LIN {X 0,Y 470.964,Z 381.158,A -85,B 0,C 180,E1 -7452.523,E2 -7452.523} C_VEL
LIN {X 0,Y 470.095,Z 393.376,A -85,B 0,C 180,E1 -7453.721,E2 -7453.721} C_VEL
LIN {X 0,Y 469.333,Z 404.5,A -85,B 0,C 180,E1 -7455.03,E2 -7455.03} C_VEL
LIN {X 0,Y 468.532,Z 415.308,A -85,B 0,C 180,E1 -7456.556,E2 -7456.556} C_VEL
LIN {X 0,Y 467.988,Z 424.27,A -85,B 0,C 180,E1 -7458.083,E2 -7458.083} C_VEL
LIN {X 0,Y 467.475,Z 431.699,A -85,B 0,C 180,E1 -7459.606,E2 -7459.606} C_VEL
LIN {X 0,Y 467.146,Z 438.641,A -85,B 0,C 180,E1 -7461.347,E2 -7461.347} C_VEL
LIN {X 0,Y 466.909,Z 444.098,A -85,B 0,C 180,E1 -7463.084,E2 -7463.084} C_VEL
LIN {X 0,Y 466.76,Z 448.219,A -85,B 0,C 180,E1 -7464.817,E2 -7464.817} C_VEL
LIN {X 0,Y 466.725,Z 451.115,A -85,B 0,C 180,E1 -7466.547,E2 -7466.547} C_VEL
LIN {X 0,Y 466.632,Z 452.862,A -85,B 0,C 180,E1 -7468.274,E2 -7468.274} C_VEL
LIN {X 0,Y 466.598,Z 453.473,A -85,B 0,C 180,E1 -7470,E2 -7470} C_VEL
LIN {X 0,Y 466.633,Z 452.914,A -85,B 0,C 180,E1 -7471.726,E2 -7471.726} C_VEL
LIN {X 0,Y 466.726,Z 451.237,A -85,B 0,C 180,E1 -7473.453,E2 -7473.453} C_VEL
LIN {X 0,Y 466.754,Z 448.408,A -85,B 0,C 180,E1 -7475.183,E2 -7475.183} C_VEL
LIN {X 0,Y 466.905,Z 444.353,A -85,B 0,C 180,E1 -7476.916,E2 -7476.916} C_VEL
LIN {X 0,Y 467.137,Z 438.975,A -85,B 0,C 180,E1 -7478.653,E2 -7478.653} C_VEL
LIN {X 0,Y 467.457,Z 432.123,A -85,B 0,C 180,E1 -7480.394,E2 -7480.394} C_VEL
LIN {X 0,Y 467.967,Z 424.747,A -85,B 0,C 180,E1 -7481.917,E2 -7481.917} C_VEL
LIN {X 0,Y 468.503,Z 415.866,A -85,B 0,C 180,E1 -7483.445,E2 -7483.445} C_VEL
LIN {X 0,Y 469.115,Z 406.807,A -85,B 0,C 180,E1 -7484.755,E2 -7484.755} C_VEL
LIN {X 0,Y 469.864,Z 396.119,A -85,B 0,C 180,E1 -7486.064,E2 -7486.064} C_VEL
LIN {X 0,Y 470.706,Z 384.762,A -85,B 0,C 180,E1 -7487.232,E2 -7487.232} C_VEL
LIN {X 0,Y 471.57,Z 371.7,A -85,B 0,C 180,E1 -7488.351,E2 -7488.351} C_VEL
LIN {X 0,Y 472.418,Z 357.63,A -85,B 0,C 180,E1 -7489.33,E2 -7489.33} C_VEL
LIN {X 0,Y 473.155,Z 344.313,A -85,B 0,C 180,E1 -7490.07,E2 -7490.07} C_VEL
LIN {X 0,Y 473.771,Z 329.352,A -85,B 0,C 180,E1 -7490.715,E2 -7490.715} C_VEL
LIN {X 0,Y 474.241,Z 315.159,A -85,B 0,C 180,E1 -7491.159,E2 -7491.159} C_VEL
LIN {X 0,Y 474.531,Z 299.207,A -85,B 0,C 180,E1 -7491.481,E2 -7491.481} C_VEL
LIN {X 0,Y 476.095,Z 164.579,A -85,B 0,C 180,E1 -7493.562,E2 -7493.562} C_VEL
LIN {X 0,Y 472.151,Z 147.036,A -85,B 0,C 180,E1 -7494.059,E2 -7494.059} C_VEL
LIN {X 0,Y 471.11,Z 143.654,A -85,B 0,C 180,E1 -7494.183,E2 -7494.183} C_VEL
LIN {X 0,Y 467.58,Z 127.87,A -85,B 0,C 180,E1 -7497.183,E2 -7497.183} C_VEL
LIN {X 0,Y 467.54,Z 127.872,A -85,B 0,C 180,E1 -7500.736,E2 -7500.736} C_VEL
LIN {X 0,Y 467.552,Z 127.869,A -85,B 0,C 180,E1 -7503.791,E2 -7503.791} C_VEL
LIN {X 0,Y 467.499,Z 127.876,A -85,B 0,C 180,E1 -7506.965,E2 -7506.965} C_VEL
LIN {X 0,Y 467.523,Z 127.868,A -85,B 0,C 180,E1 -7509.946,E2 -7509.946} C_VEL
LIN {X 0,Y 467.517,Z 127.874,A -85,B 0,C 180,E1 -7512.568,E2 -7512.568} C_VEL
LIN {X 0,Y 467.563,Z 127.872,A -85,B 0,C 180,E1 -7515.052,E2 -7515.052} C_VEL
LIN {X 0,Y 467.561,Z 127.864,A -85,B 0,C 180,E1 -7518.726,E2 -7518.726} C_VEL
LIN {X 0,Y 467.542,Z 127.863,A -85,B 0,C 180,E1 -7521.953,E2 -7521.953} C_VEL
LIN {X 0,Y 467.552,Z 127.869,A -85,B 0,C 180,E1 -7525.166,E2 -7525.166} C_VEL
LIN {X 0,Y 467.551,Z 127.861,A -85,B 0,C 180,E1 -7528.257,E2 -7528.257} C_VEL
LIN {X 0,Y 467.526,Z 127.869,A -85,B 0,C 180,E1 -7531.247,E2 -7531.247} C_VEL
LIN {X 0,Y 467.58,Z 127.866,A -85,B 0,C 180,E1 -7534.401,E2 -7534.401} C_VEL
LIN {X 0,Y 467.57,Z 127.862,A -85,B 0,C 180,E1 -7536.995,E2 -7536.995} C_VEL
LIN {X 0,Y 467.613,Z 127.861,A -85,B 0,C 180,E1 -7539.777,E2 -7539.777} C_VEL
LIN {X 0,Y 467.568,Z 127.867,A -85,B 0,C 180,E1 -7542.505,E2 -7542.505} C_VEL
LIN {X 0,Y 467.597,Z 127.86,A -85,B 0,C 180,E1 -7545.196,E2 -7545.196} C_VEL
LIN {X 0,Y 467.66,Z 127.857,A -85,B 0,C 180,E1 -7547.855,E2 -7547.855} C_VEL
LIN {X 0,Y 467.66,Z 127.849,A -85,B 0,C 180,E1 -7551.357,E2 -7551.357} C_VEL
LIN {X 0,Y 467.706,Z 127.85,A -85,B 0,C 180,E1 -7553.962,E2 -7553.962} C_VEL
LIN {X 0,Y 467.816,Z 127.836,A -85,B 0,C 180,E1 -7557.417,E2 -7557.417} C_VEL
LIN {X 0,Y 467.855,Z 127.828,A -85,B 0,C 180,E1 -7560,E2 -7560} C_VEL
LIN {X 0,Y 467.852,Z 127.829,A -85,B 0,C 180,E1 -7562.583,E2 -7562.583} C_VEL
LIN {X 0,Y 467.715,Z 127.847,A -85,B 0,C 180,E1 -7566.038,E2 -7566.038} C_VEL
LIN {X 0,Y 467.67,Z 127.85,A -85,B 0,C 180,E1 -7568.643,E2 -7568.643} C_VEL
LIN {X 0,Y 467.659,Z 127.853,A -85,B 0,C 180,E1 -7572.145,E2 -7572.145} C_VEL
LIN {X 0,Y 467.651,Z 127.856,A -85,B 0,C 180,E1 -7575.884,E2 -7575.884} C_VEL
LIN {X 0,Y 467.624,Z 127.864,A -85,B 0,C 180,E1 -7579.308,E2 -7579.308} C_VEL
LIN {X 0,Y 467.536,Z 127.866,A -85,B 0,C 180,E1 -7582.074,E2 -7582.074} C_VEL
LIN {X 0,Y 467.57,Z 127.871,A -85,B 0,C 180,E1 -7584.889,E2 -7584.889} C_VEL
LIN {X 0,Y 467.582,Z 127.863,A -85,B 0,C 180,E1 -7587.771,E2 -7587.771} C_VEL
LIN {X 0,Y 467.569,Z 127.868,A -85,B 0,C 180,E1 -7591.044,E2 -7591.044} C_VEL
LIN {X 0,Y 467.579,Z 127.862,A -85,B 0,C 180,E1 -7594.24,E2 -7594.24} C_VEL
LIN {X 0,Y 467.549,Z 127.867,A -85,B 0,C 180,E1 -7597.186,E2 -7597.186} C_VEL
LIN {X 0,Y 467.576,Z 127.866,A -85,B 0,C 180,E1 -7600.265,E2 -7600.265} C_VEL
LIN {X 0,Y 467.588,Z 127.866,A -85,B 0,C 180,E1 -7602.567,E2 -7602.567} C_VEL
LIN {X 0,Y 467.567,Z 127.865,A -85,B 0,C 180,E1 -7605.052,E2 -7605.052} C_VEL
LIN {X 0,Y 467.59,Z 127.861,A -85,B 0,C 180,E1 -7607.44,E2 -7607.44} C_VEL
LIN {X 0,Y 467.583,Z 127.863,A -85,B 0,C 180,E1 -7610.855,E2 -7610.855} C_VEL
LIN {X 0,Y 467.561,Z 127.871,A -85,B 0,C 180,E1 -7614.261,E2 -7614.261} C_VEL
LIN {X 0,Y 467.583,Z 127.866,A -85,B 0,C 180,E1 -7617.321,E2 -7617.321} C_VEL
LIN {X 0,Y 467.577,Z 127.992,A -85,B 0,C 180,E1 -7619.641,E2 -7619.641} C_VEL
LIN {X 0,Y 471.398,Z 143.466,A -85,B 0,C 180,E1 -7622.297,E2 -7622.297} C_VEL
LIN {X 0,Y 472.18,Z 147.627,A -85,B 0,C 180,E1 -7622.979,E2 -7622.979} C_VEL
LIN {X 0,Y 471.23,Z 165.357,A -85,B 0,C 180,E1 -7625.608,E2 -7625.608} C_VEL
LIN {X 0,Y 471.125,Z 167.06,A -85,B 0,C 180,E1 -7625.858,E2 -7625.858} C_VEL
LIN {X 0,Y 475.883,Z 191.887,A -85,B 0,C 180,E1 -7626.518,E2 -7626.518} C_VEL
LIN {X 0,Y 474.175,Z 334.044,A -85,B 0,C 180,E1 -7628.736,E2 -7628.736} C_VEL
LIN {X 0,Y 473.612,Z 349.775,A -85,B 0,C 180,E1 -7629.159,E2 -7629.159} C_VEL
LIN {X 0,Y 473.059,Z 363.831,A -85,B 0,C 180,E1 -7629.704,E2 -7629.704} C_VEL
LIN {X 0,Y 472.272,Z 378.294,A -85,B 0,C 180,E1 -7630.438,E2 -7630.438} C_VEL
LIN {X 0,Y 471.417,Z 391.803,A -85,B 0,C 180,E1 -7631.305,E2 -7631.305} C_VEL
LIN {X 0,Y 470.502,Z 405.559,A -85,B 0,C 180,E1 -7632.393,E2 -7632.393} C_VEL
LIN {X 0,Y 469.702,Z 418.015,A -85,B 0,C 180,E1 -7633.595,E2 -7633.595} C_VEL
LIN {X 0,Y 468.789,Z 430.23,A -85,B 0,C 180,E1 -7635.012,E2 -7635.012} C_VEL
LIN {X 0,Y 468.08,Z 441.095,A -85,B 0,C 180,E1 -7636.542,E2 -7636.542} C_VEL
LIN {X 0,Y 467.611,Z 450.148,A -85,B 0,C 180,E1 -7638.073,E2 -7638.073} C_VEL
LIN {X 0,Y 467.228,Z 457.657,A -85,B 0,C 180,E1 -7639.601,E2 -7639.601} C_VEL
LIN {X 0,Y 466.908,Z 464.664,A -85,B 0,C 180,E1 -7641.343,E2 -7641.343} C_VEL
LIN {X 0,Y 466.818,Z 470.178,A -85,B 0,C 180,E1 -7643.082,E2 -7643.082} C_VEL
LIN {X 0,Y 466.685,Z 474.344,A -85,B 0,C 180,E1 -7644.816,E2 -7644.816} C_VEL
LIN {X 0,Y 466.634,Z 477.265,A -85,B 0,C 180,E1 -7646.546,E2 -7646.546} C_VEL
LIN {X 0,Y 466.604,Z 479.007,A -85,B 0,C 180,E1 -7648.274,E2 -7648.274} C_VEL
LIN {X 0,Y 466.596,Z 479.605,A -85,B 0,C 180,E1 -7650,E2 -7650} C_VEL
LIN {X 0,Y 466.604,Z 479.005,A -85,B 0,C 180,E1 -7651.726,E2 -7651.726} C_VEL
LIN {X 0,Y 466.634,Z 477.259,A -85,B 0,C 180,E1 -7653.454,E2 -7653.454} C_VEL
LIN {X 0,Y 466.686,Z 474.34,A -85,B 0,C 180,E1 -7655.184,E2 -7655.184} C_VEL
LIN {X 0,Y 466.818,Z 470.179,A -85,B 0,C 180,E1 -7656.918,E2 -7656.918} C_VEL
LIN {X 0,Y 466.908,Z 464.662,A -85,B 0,C 180,E1 -7658.657,E2 -7658.657} C_VEL
LIN {X 0,Y 467.227,Z 457.646,A -85,B 0,C 180,E1 -7660.399,E2 -7660.399} C_VEL
LIN {X 0,Y 467.608,Z 450.138,A -85,B 0,C 180,E1 -7661.927,E2 -7661.927} C_VEL
LIN {X 0,Y 468.08,Z 441.088,A -85,B 0,C 180,E1 -7663.458,E2 -7663.458} C_VEL
LIN {X 0,Y 468.789,Z 430.218,A -85,B 0,C 180,E1 -7664.988,E2 -7664.988} C_VEL
LIN {X 0,Y 469.675,Z 418.004,A -85,B 0,C 180,E1 -7666.406,E2 -7666.406} C_VEL
LIN {X 0,Y 470.499,Z 405.548,A -85,B 0,C 180,E1 -7667.607,E2 -7667.607} C_VEL
LIN {X 0,Y 471.406,Z 391.772,A -85,B 0,C 180,E1 -7668.695,E2 -7668.695} C_VEL
LIN {X 0,Y 472.268,Z 378.248,A -85,B 0,C 180,E1 -7669.562,E2 -7669.562} C_VEL
LIN {X 0,Y 473.057,Z 363.696,A -85,B 0,C 180,E1 -7670.301,E2 -7670.301} C_VEL
LIN {X 0,Y 473.673,Z 349.107,A -85,B 0,C 180,E1 -7670.861,E2 -7670.861} C_VEL
LIN {X 0,Y 474.164,Z 333.95,A -85,B 0,C 180,E1 -7671.264,E2 -7671.264} C_VEL
LIN {X 0,Y 475.8,Z 200.78,A -85,B 0,C 180,E1 -7673.34,E2 -7673.34} C_VEL
LIN {X 0,Y 475.737,Z 190.572,A -85,B 0,C 180,E1 -7673.507,E2 -7673.507} C_VEL
LIN {X 0,Y 471.132,Z 167.042,A -85,B 0,C 180,E1 -7674.14,E2 -7674.14} C_VEL
LIN {X 0,Y 472.175,Z 147.582,A -85,B 0,C 180,E1 -7677.024,E2 -7677.024} C_VEL
LIN {X 0,Y 469.786,Z 136.715,A -85,B 0,C 180,E1 -7678.839,E2 -7678.839} C_VEL
LIN {X 0,Y 467.58,Z 127.866,A -85,B 0,C 180,E1 -7680.389,E2 -7680.389} C_VEL
LIN {X 0,Y 467.587,Z 127.862,A -85,B 0,C 180,E1 -7683.788,E2 -7683.788} C_VEL
LIN {X 0,Y 467.549,Z 127.868,A -85,B 0,C 180,E1 -7687.186,E2 -7687.186} C_VEL
LIN {X 0,Y 467.578,Z 127.865,A -85,B 0,C 180,E1 -7690.265,E2 -7690.265} C_VEL
LIN {X 0,Y 467.587,Z 127.861,A -85,B 0,C 180,E1 -7692.567,E2 -7692.567} C_VEL
LIN {X 0,Y 467.567,Z 127.864,A -85,B 0,C 180,E1 -7695.053,E2 -7695.053} C_VEL
LIN {X 0,Y 467.59,Z 127.865,A -85,B 0,C 180,E1 -7697.44,E2 -7697.44} C_VEL
LIN {X 0,Y 467.561,Z 127.866,A -85,B 0,C 180,E1 -7700.853,E2 -7700.853} C_VEL
LIN {X 0,Y 467.56,Z 127.862,A -85,B 0,C 180,E1 -7704.261,E2 -7704.261} C_VEL
LIN {X 0,Y 467.581,Z 127.865,A -85,B 0,C 180,E1 -7707.322,E2 -7707.322} C_VEL
LIN {X 0,Y 467.57,Z 127.863,A -85,B 0,C 180,E1 -7710.668,E2 -7710.668} C_VEL
LIN {X 0,Y 467.588,Z 127.865,A -85,B 0,C 180,E1 -7713.198,E2 -7713.198} C_VEL
LIN {X 0,Y 467.591,Z 127.861,A -85,B 0,C 180,E1 -7716.47,E2 -7716.47} C_VEL
LIN {X 0,Y 467.623,Z 127.854,A -85,B 0,C 180,E1 -7719.777,E2 -7719.777} C_VEL
LIN {X 0,Y 467.597,Z 127.864,A -85,B 0,C 180,E1 -7722.506,E2 -7722.506} C_VEL
LIN {X 0,Y 467.605,Z 127.863,A -85,B 0,C 180,E1 -7725.197,E2 -7725.197} C_VEL
LIN {X 0,Y 467.659,Z 127.849,A -85,B 0,C 180,E1 -7727.855,E2 -7727.855} C_VEL
LIN {X 0,Y 467.67,Z 127.848,A -85,B 0,C 180,E1 -7731.357,E2 -7731.357} C_VEL
LIN {X 0,Y 467.715,Z 127.847,A -85,B 0,C 180,E1 -7733.962,E2 -7733.962} C_VEL
LIN {X 0,Y 467.852,Z 127.828,A -85,B 0,C 180,E1 -7737.417,E2 -7737.417} C_VEL
LIN {X 0,Y 467.855,Z 127.83,A -85,B 0,C 180,E1 -7740,E2 -7740} C_VEL
LIN {X 0,Y 467.817,Z 127.837,A -85,B 0,C 180,E1 -7742.583,E2 -7742.583} C_VEL
LIN {X 0,Y 467.712,Z 127.849,A -85,B 0,C 180,E1 -7746.038,E2 -7746.038} C_VEL
LIN {X 0,Y 467.66,Z 127.851,A -85,B 0,C 180,E1 -7748.643,E2 -7748.643} C_VEL
LIN {X 0,Y 467.659,Z 127.856,A -85,B 0,C 180,E1 -7752.145,E2 -7752.145} C_VEL
LIN {X 0,Y 467.615,Z 127.863,A -85,B 0,C 180,E1 -7755.696,E2 -7755.696} C_VEL
LIN {X 0,Y 467.62,Z 127.859,A -85,B 0,C 180,E1 -7759.308,E2 -7759.308} C_VEL
LIN {X 0,Y 467.535,Z 127.873,A -85,B 0,C 180,E1 -7762.074,E2 -7762.074} C_VEL
LIN {X 0,Y 467.561,Z 127.862,A -85,B 0,C 180,E1 -7764.89,E2 -7764.89} C_VEL
LIN {X 0,Y 467.547,Z 127.865,A -85,B 0,C 180,E1 -7767.774,E2 -7767.774} C_VEL
LIN {X 0,Y 467.549,Z 127.868,A -85,B 0,C 180,E1 -7771.04,E2 -7771.04} C_VEL
LIN {X 0,Y 467.577,Z 127.86,A -85,B 0,C 180,E1 -7774.24,E2 -7774.24} C_VEL
LIN {X 0,Y 467.539,Z 127.871,A -85,B 0,C 180,E1 -7777.184,E2 -7777.184} C_VEL
LIN {X 0,Y 467.557,Z 127.864,A -85,B 0,C 180,E1 -7780.267,E2 -7780.267} C_VEL
LIN {X 0,Y 467.545,Z 127.867,A -85,B 0,C 180,E1 -7783.746,E2 -7783.746} C_VEL
LIN {X 0,Y 467.545,Z 127.867,A -85,B 0,C 180,E1 -7786.254,E2 -7786.254} C_VEL
LIN {X 0,Y 467.556,Z 127.868,A -85,B 0,C 180,E1 -7789.733,E2 -7789.733} C_VEL
LIN {X 0,Y 467.517,Z 127.877,A -85,B 0,C 180,E1 -7792.819,E2 -7792.819} C_VEL
LIN {X 0,Y 467.565,Z 127.867,A -85,B 0,C 180,E1 -7795.762,E2 -7795.762} C_VEL
LIN {X 0,Y 467.527,Z 127.867,A -85,B 0,C 180,E1 -7798.964,E2 -7798.964} C_VEL
LIN {X 0,Y 467.538,Z 127.873,A -85,B 0,C 180,E1 -7802.226,E2 -7802.226} C_VEL
LIN {X 0,Y 467.586,Z 127.922,A -85,B 0,C 180,E1 -7802.927,E2 -7802.927} C_VEL
LIN {X 0,Y 470.737,Z 142.01,A -85,B 0,C 180,E1 -7805.605,E2 -7805.605} C_VEL
LIN {X 0,Y 471.126,Z 143.896,A -85,B 0,C 180,E1 -7805.927,E2 -7805.927} C_VEL
LIN {X 0,Y 472.934,Z 150.367,A -85,B 0,C 180,E1 -7806.132,E2 -7806.132} C_VEL
LIN {X 0,Y 476.111,Z 164.515,A -85,B 0,C 180,E1 -7806.531,E2 -7806.531} C_VEL
LIN {X 0,Y 475.725,Z 202.904,A -85,B 0,C 180,E1 -7807.129,E2 -7807.129} C_VEL
LIN {X 0,Y 475.079,Z 208.751,A -85,B 0,C 180,E1 -7807.19,E2 -7807.19} C_VEL
LIN {X 0,Y 469.531,Z 227.805,A -85,B 0,C 180,E1 -7807.213,E2 -7807.213} C_VEL
LIN {X 0,Y 468.741,Z 233.659,A -85,B 0,C 180,E1 -7807.267,E2 -7807.267} C_VEL
LIN {X 0,Y 467.779,Z 308.963,A -85,B 0,C 180,E1 -7808.466,E2 -7808.466} C_VEL
LIN {X 0,Y 467.327,Z 324.475,A -85,B 0,C 180,E1 -7808.887,E2 -7808.887} C_VEL
LIN {X 0,Y 466.807,Z 338.824,A -85,B 0,C 180,E1 -7809.451,E2 -7809.451} C_VEL
LIN {X 0,Y 466.013,Z 352.734,A -85,B 0,C 180,E1 -7810.164,E2 -7810.164} C_VEL
LIN {X 0,Y 465.186,Z 366.326,A -85,B 0,C 180,E1 -7811.045,E2 -7811.045} C_VEL
LIN {X 0,Y 464.329,Z 378.821,A -85,B 0,C 180,E1 -7812.038,E2 -7812.038} C_VEL
LIN {X 0,Y 463.397,Z 391.471,A -85,B 0,C 180,E1 -7813.252,E2 -7813.252} C_VEL
LIN {X 0,Y 462.548,Z 402.936,A -85,B 0,C 180,E1 -7814.58,E2 -7814.58} C_VEL
LIN {X 0,Y 461.825,Z 412.582,A -85,B 0,C 180,E1 -7815.908,E2 -7815.908} C_VEL
LIN {X 0,Y 461.063,Z 422.108,A -85,B 0,C 180,E1 -7817.468,E2 -7817.468} C_VEL
LIN {X 0,Y 460.627,Z 429.9,A -85,B 0,C 180,E1 -7819.005,E2 -7819.005} C_VEL
LIN {X 0,Y 460.165,Z 437.243,A -85,B 0,C 180,E1 -7820.772,E2 -7820.772} C_VEL
LIN {X 0,Y 459.9,Z 443.069,A -85,B 0,C 180,E1 -7822.537,E2 -7822.537} C_VEL
LIN {X 0,Y 459.817,Z 446.516,A -85,B 0,C 180,E1 -7823.858,E2 -7823.858} C_VEL
LIN {X 0,Y 459.595,Z 450.016,A -85,B 0,C 180,E1 -7825.615,E2 -7825.615} C_VEL
LIN {X 0,Y 459.6,Z 452.328,A -85,B 0,C 180,E1 -7827.371,E2 -7827.371} C_VEL
LIN {X 0,Y 459.521,Z 453.514,A -85,B 0,C 180,E1 -7829.124,E2 -7829.124} C_VEL
LIN {X 0,Y 459.521,Z 453.531,A -85,B 0,C 180,E1 -7830.876,E2 -7830.876} C_VEL
LIN {X 0,Y 459.601,Z 452.415,A -85,B 0,C 180,E1 -7832.629,E2 -7832.629} C_VEL
LIN {X 0,Y 459.594,Z 450.171,A -85,B 0,C 180,E1 -7834.385,E2 -7834.385} C_VEL
LIN {X 0,Y 459.787,Z 446.735,A -85,B 0,C 180,E1 -7836.142,E2 -7836.142} C_VEL
LIN {X 0,Y 459.965,Z 442.035,A -85,B 0,C 180,E1 -7837.904,E2 -7837.904} C_VEL
LIN {X 0,Y 460.255,Z 435.944,A -85,B 0,C 180,E1 -7839.67,E2 -7839.67} C_VEL
LIN {X 0,Y 460.814,Z 428.268,A -85,B 0,C 180,E1 -7841.436,E2 -7841.436} C_VEL
LIN {X 0,Y 461.285,Z 420.112,A -85,B 0,C 180,E1 -7842.983,E2 -7842.983} C_VEL
LIN {X 0,Y 461.986,Z 410.229,A -85,B 0,C 180,E1 -7844.537,E2 -7844.537} C_VEL
LIN {X 0,Y 462.757,Z 400.117,A -85,B 0,C 180,E1 -7845.865,E2 -7845.865} C_VEL
LIN {X 0,Y 463.621,Z 389.042,A -85,B 0,C 180,E1 -7847.09,E2 -7847.09} C_VEL
LIN {X 0,Y 464.406,Z 377.289,A -85,B 0,C 180,E1 -7848.187,E2 -7848.187} C_VEL
LIN {X 0,Y 465.322,Z 364.457,A -85,B 0,C 180,E1 -7849.178,E2 -7849.178} C_VEL
LIN {X 0,Y 466.18,Z 350.381,A -85,B 0,C 180,E1 -7850.058,E2 -7850.058} C_VEL
LIN {X 0,Y 466.925,Z 335.079,A -85,B 0,C 180,E1 -7850.802,E2 -7850.802} C_VEL
LIN {X 0,Y 467.481,Z 319.758,A -85,B 0,C 180,E1 -7851.349,E2 -7851.349} C_VEL
LIN {X 0,Y 467.889,Z 304.527,A -85,B 0,C 180,E1 -7851.708,E2 -7851.708} C_VEL
LIN {X 0,Y 469.572,Z 164.991,A -85,B 0,C 180,E1 -7853.906,E2 -7853.906} C_VEL
LIN {X 0,Y 465.333,Z 147.428,A -85,B 0,C 180,E1 -7854.431,E2 -7854.431} C_VEL
LIN {X 0,Y 463.967,Z 143.875,A -85,B 0,C 180,E1 -7854.577,E2 -7854.577} C_VEL
LIN {X 0,Y 460.858,Z 130.147,A -85,B 0,C 180,E1 -7857.226,E2 -7857.226} C_VEL
LIN {X 0,Y 460.511,Z 128.75,A -85,B 0,C 180,E1 -7857.527,E2 -7857.527} C_VEL
LIN {X 0,Y 460.479,Z 128.751,A -85,B 0,C 180,E1 -7860.243,E2 -7860.243} C_VEL
LIN {X 0,Y 460.501,Z 128.751,A -85,B 0,C 180,E1 -7863.327,E2 -7863.327} C_VEL
LIN {X 0,Y 460.455,Z 128.752,A -85,B 0,C 180,E1 -7866.532,E2 -7866.532} C_VEL
LIN {X 0,Y 460.475,Z 128.746,A -85,B 0,C 180,E1 -7869.869,E2 -7869.869} C_VEL
LIN {X 0,Y 460.457,Z 128.756,A -85,B 0,C 180,E1 -7872.893,E2 -7872.893} C_VEL
LIN {X 0,Y 460.495,Z 128.746,A -85,B 0,C 180,E1 -7875.833,E2 -7875.833} C_VEL
LIN {X 0,Y 460.515,Z 128.746,A -85,B 0,C 180,E1 -7878.987,E2 -7878.987} C_VEL
LIN {X 0,Y 460.484,Z 128.742,A -85,B 0,C 180,E1 -7882.375,E2 -7882.375} C_VEL
LIN {X 0,Y 460.535,Z 128.741,A -85,B 0,C 180,E1 -7885.623,E2 -7885.623} C_VEL
LIN {X 0,Y 460.506,Z 128.735,A -85,B 0,C 180,E1 -7888.742,E2 -7888.742} C_VEL
LIN {X 0,Y 460.498,Z 128.745,A -85,B 0,C 180,E1 -7891.763,E2 -7891.763} C_VEL
LIN {X 0,Y 460.524,Z 128.745,A -85,B 0,C 180,E1 -7894.703,E2 -7894.703} C_VEL
LIN {X 0,Y 460.505,Z 128.742,A -85,B 0,C 180,E1 -7897.571,E2 -7897.571} C_VEL
LIN {X 0,Y 460.564,Z 128.74,A -85,B 0,C 180,E1 -7900.384,E2 -7900.384} C_VEL
LIN {X 0,Y 460.569,Z 128.743,A -85,B 0,C 180,E1 -7904.058,E2 -7904.058} C_VEL
LIN {X 0,Y 460.613,Z 128.732,A -85,B 0,C 180,E1 -7907.666,E2 -7907.666} C_VEL
LIN {X 0,Y 460.612,Z 128.726,A -85,B 0,C 180,E1 -7911.223,E2 -7911.223} C_VEL
LIN {X 0,Y 460.672,Z 128.728,A -85,B 0,C 180,E1 -7913.869,E2 -7913.869} C_VEL
LIN {X 0,Y 460.76,Z 128.715,A -85,B 0,C 180,E1 -7917.377,E2 -7917.377} C_VEL
LIN {X 0,Y 460.825,Z 128.704,A -85,B 0,C 180,E1 -7920,E2 -7920} C_VEL
LIN {X 0,Y 460.792,Z 128.708,A -85,B 0,C 180,E1 -7922.622,E2 -7922.622} C_VEL
LIN {X 0,Y 460.68,Z 128.723,A -85,B 0,C 180,E1 -7926.13,E2 -7926.13} C_VEL
LIN {X 0,Y 460.62,Z 128.729,A -85,B 0,C 180,E1 -7928.776,E2 -7928.776} C_VEL
LIN {X 0,Y 460.612,Z 128.731,A -85,B 0,C 180,E1 -7932.334,E2 -7932.334} C_VEL
LIN {X 0,Y 460.603,Z 128.733,A -85,B 0,C 180,E1 -7935.997,E2 -7935.997} C_VEL
LIN {X 0,Y 460.57,Z 128.739,A -85,B 0,C 180,E1 -7939.615,E2 -7939.615} C_VEL
LIN {X 0,Y 460.512,Z 128.743,A -85,B 0,C 180,E1 -7942.428,E2 -7942.428} C_VEL
LIN {X 0,Y 460.549,Z 128.737,A -85,B 0,C 180,E1 -7945.796,E2 -7945.796} C_VEL
LIN {X 0,Y 460.529,Z 128.743,A -85,B 0,C 180,E1 -7948.234,E2 -7948.234} C_VEL
LIN {X 0,Y 460.522,Z 128.744,A -85,B 0,C 180,E1 -7951.283,E2 -7951.283} C_VEL
LIN {X 0,Y 460.525,Z 128.743,A -85,B 0,C 180,E1 -7954.504,E2 -7954.504} C_VEL
LIN {X 0,Y 460.502,Z 128.743,A -85,B 0,C 180,E1 -7957.623,E2 -7957.623} C_VEL
LIN {X 0,Y 460.54,Z 128.742,A -85,B 0,C 180,E1 -7960.269,E2 -7960.269} C_VEL
LIN {X 0,Y 460.5,Z 128.746,A -85,B 0,C 180,E1 -7963.375,E2 -7963.375} C_VEL
LIN {X 0,Y 460.5,Z 128.747,A -85,B 0,C 180,E1 -7966.624,E2 -7966.624} C_VEL
LIN {X 0,Y 460.543,Z 128.735,A -85,B 0,C 180,E1 -7969.73,E2 -7969.73} C_VEL
LIN {X 0,Y 460.501,Z 128.748,A -85,B 0,C 180,E1 -7972.524,E2 -7972.524} C_VEL
LIN {X 0,Y 460.547,Z 128.744,A -85,B 0,C 180,E1 -7975.624,E2 -7975.624} C_VEL
LIN {X 0,Y 460.538,Z 128.744,A -85,B 0,C 180,E1 -7978.744,E2 -7978.744} C_VEL
LIN {X 0,Y 460.534,Z 128.783,A -85,B 0,C 180,E1 -7979.286,E2 -7979.286} C_VEL
LIN {X 0,Y 464.382,Z 144.41,A -85,B 0,C 180,E1 -7982.02,E2 -7982.02} C_VEL
LIN {X 0,Y 465.346,Z 149.156,A -85,B 0,C 180,E1 -7982.816,E2 -7982.816} C_VEL
LIN {X 0,Y 464.468,Z 165.058,A -85,B 0,C 180,E1 -7985.213,E2 -7985.213} C_VEL
LIN {X 0,Y 464.367,Z 166.838,A -85,B 0,C 180,E1 -7985.481,E2 -7985.481} C_VEL
LIN {X 0,Y 469.365,Z 192.662,A -85,B 0,C 180,E1 -7986.188,E2 -7986.188} C_VEL
LIN {X 0,Y 467.572,Z 333.856,A -85,B 0,C 180,E1 -7988.421,E2 -7988.421} C_VEL
LIN {X 0,Y 466.98,Z 349.574,A -85,B 0,C 180,E1 -7988.849,E2 -7988.849} C_VEL
LIN {X 0,Y 466.363,Z 364.228,A -85,B 0,C 180,E1 -7989.428,E2 -7989.428} C_VEL
LIN {X 0,Y 465.545,Z 378.099,A -85,B 0,C 180,E1 -7990.143,E2 -7990.143} C_VEL
LIN {X 0,Y 464.669,Z 391.607,A -85,B 0,C 180,E1 -7991.023,E2 -7991.023} C_VEL
LIN {X 0,Y 463.678,Z 405.362,A -85,B 0,C 180,E1 -7992.126,E2 -7992.126} C_VEL
LIN {X 0,Y 462.833,Z 417.817,A -85,B 0,C 180,E1 -7993.345,E2 -7993.345} C_VEL
LIN {X 0,Y 461.857,Z 430.031,A -85,B 0,C 180,E1 -7994.782,E2 -7994.782} C_VEL
LIN {X 0,Y 461.119,Z 440.896,A -85,B 0,C 180,E1 -7996.335,E2 -7996.335} C_VEL
LIN {X 0,Y 460.591,Z 449.948,A -85,B 0,C 180,E1 -7997.889,E2 -7997.889} C_VEL
LIN {X 0,Y 460.216,Z 457.458,A -85,B 0,C 180,E1 -7999.441,E2 -7999.441} C_VEL
LIN {X 0,Y 459.851,Z 464.465,A -85,B 0,C 180,E1 -8001.209,E2 -8001.209} C_VEL
LIN {X 0,Y 459.727,Z 469.978,A -85,B 0,C 180,E1 -8002.975,E2 -8002.975} C_VEL
LIN {X 0,Y 459.595,Z 474.145,A -85,B 0,C 180,E1 -8004.736,E2 -8004.736} C_VEL
LIN {X 0,Y 459.53,Z 477.066,A -85,B 0,C 180,E1 -8006.493,E2 -8006.493} C_VEL
LIN {X 0,Y 459.517,Z 478.809,A -85,B 0,C 180,E1 -8008.247,E2 -8008.247} C_VEL
LIN {X 0,Y 459.527,Z 479.407,A -85,B 0,C 180,E1 -8010,E2 -8010} C_VEL
LIN {X 0,Y 459.517,Z 478.806,A -85,B 0,C 180,E1 -8011.753,E2 -8011.753} C_VEL
LIN {X 0,Y 459.53,Z 477.059,A -85,B 0,C 180,E1 -8013.507,E2 -8013.507} C_VEL
LIN {X 0,Y 459.598,Z 474.14,A -85,B 0,C 180,E1 -8015.264,E2 -8015.264} C_VEL
LIN {X 0,Y 459.727,Z 469.979,A -85,B 0,C 180,E1 -8017.025,E2 -8017.025} C_VEL
LIN {X 0,Y 459.851,Z 464.461,A -85,B 0,C 180,E1 -8018.791,E2 -8018.791} C_VEL
LIN {X 0,Y 460.214,Z 457.445,A -85,B 0,C 180,E1 -8020.559,E2 -8020.559} C_VEL
LIN {X 0,Y 460.584,Z 449.936,A -85,B 0,C 180,E1 -8022.111,E2 -8022.111} C_VEL
LIN {X 0,Y 461.119,Z 440.886,A -85,B 0,C 180,E1 -8023.665,E2 -8023.665} C_VEL
LIN {X 0,Y 461.855,Z 430.015,A -85,B 0,C 180,E1 -8025.218,E2 -8025.218} C_VEL
LIN {X 0,Y 462.811,Z 417.801,A -85,B 0,C 180,E1 -8026.656,E2 -8026.656} C_VEL
LIN {X 0,Y 463.679,Z 405.345,A -85,B 0,C 180,E1 -8027.874,E2 -8027.874} C_VEL
LIN {X 0,Y 464.644,Z 391.568,A -85,B 0,C 180,E1 -8028.978,E2 -8028.978} C_VEL
LIN {X 0,Y 465.533,Z 378.043,A -85,B 0,C 180,E1 -8029.857,E2 -8029.857} C_VEL
LIN {X 0,Y 466.352,Z 364.112,A -85,B 0,C 180,E1 -8030.576,E2 -8030.576} C_VEL
LIN {X 0,Y 467.051,Z 348.901,A -85,B 0,C 180,E1 -8031.17,E2 -8031.17} C_VEL
LIN {X 0,Y 467.556,Z 333.74,A -85,B 0,C 180,E1 -8031.58,E2 -8031.58} C_VEL
LIN {X 0,Y 469.117,Z 211.55,A -85,B 0,C 180,E1 -8033.513,E2 -8033.513} C_VEL
LIN {X 0,Y 469.296,Z 191.977,A -85,B 0,C 180,E1 -8033.823,E2 -8033.823} C_VEL
LIN {X 0,Y 464.378,Z 166.694,A -85,B 0,C 180,E1 -8034.535,E2 -8034.535} C_VEL
LIN {X 0,Y 465.34,Z 149.118,A -85,B 0,C 180,E1 -8037.185,E2 -8037.185} C_VEL
LIN {X 0,Y 462.31,Z 135.727,A -85,B 0,C 180,E1 -8039.474,E2 -8039.474} C_VEL
LIN {X 0,Y 460.547,Z 128.742,A -85,B 0,C 180,E1 -8040.745,E2 -8040.745} C_VEL
LIN {X 0,Y 460.53,Z 128.736,A -85,B 0,C 180,E1 -8043.325,E2 -8043.325} C_VEL
LIN {X 0,Y 460.477,Z 128.75,A -85,B 0,C 180,E1 -8046.53,E2 -8046.53} C_VEL
LIN {X 0,Y 460.559,Z 128.744,A -85,B 0,C 180,E1 -8049.86,E2 -8049.86} C_VEL
LIN {X 0,Y 460.513,Z 128.743,A -85,B 0,C 180,E1 -8052.9,E2 -8052.9} C_VEL
LIN {X 0,Y 460.51,Z 128.748,A -85,B 0,C 180,E1 -8055.831,E2 -8055.831} C_VEL
LIN {X 0,Y 460.531,Z 128.742,A -85,B 0,C 180,E1 -8058.989,E2 -8058.989} C_VEL
LIN {X 0,Y 460.52,Z 128.746,A -85,B 0,C 180,E1 -8061.266,E2 -8061.266} C_VEL
LIN {X 0,Y 460.509,Z 128.74,A -85,B 0,C 180,E1 -8064.554,E2 -8064.554} C_VEL
LIN {X 0,Y 460.531,Z 128.743,A -85,B 0,C 180,E1 -8067.716,E2 -8067.716} C_VEL
LIN {X 0,Y 460.539,Z 128.739,A -85,B 0,C 180,E1 -8070.769,E2 -8070.769} C_VEL
LIN {X 0,Y 460.543,Z 128.74,A -85,B 0,C 180,E1 -8073.734,E2 -8073.734} C_VEL
LIN {X 0,Y 460.545,Z 128.74,A -85,B 0,C 180,E1 -8076.624,E2 -8076.624} C_VEL
LIN {X 0,Y 460.552,Z 128.737,A -85,B 0,C 180,E1 -8079.453,E2 -8079.453} C_VEL
LIN {X 0,Y 460.549,Z 128.74,A -85,B 0,C 180,E1 -8082.23,E2 -8082.23} C_VEL
LIN {X 0,Y 460.565,Z 128.743,A -85,B 0,C 180,E1 -8084.965,E2 -8084.965} C_VEL
LIN {X 0,Y 460.612,Z 128.727,A -85,B 0,C 180,E1 -8087.666,E2 -8087.666} C_VEL
LIN {X 0,Y 460.62,Z 128.727,A -85,B 0,C 180,E1 -8091.224,E2 -8091.224} C_VEL
LIN {X 0,Y 460.68,Z 128.723,A -85,B 0,C 180,E1 -8093.87,E2 -8093.87} C_VEL
LIN {X 0,Y 460.793,Z 128.708,A -85,B 0,C 180,E1 -8097.378,E2 -8097.378} C_VEL
LIN {X 0,Y 460.824,Z 128.705,A -85,B 0,C 180,E1 -8100,E2 -8100} C_VEL
LIN {X 0,Y 460.761,Z 128.715,A -85,B 0,C 180,E1 -8102.623,E2 -8102.623} C_VEL
LIN {X 0,Y 460.677,Z 128.727,A -85,B 0,C 180,E1 -8106.13,E2 -8106.13} C_VEL
LIN {X 0,Y 460.612,Z 128.728,A -85,B 0,C 180,E1 -8108.777,E2 -8108.777} C_VEL
LIN {X 0,Y 460.612,Z 128.731,A -85,B 0,C 180,E1 -8112.334,E2 -8112.334} C_VEL
LIN {X 0,Y 460.559,Z 128.742,A -85,B 0,C 180,E1 -8115.978,E2 -8115.978} C_VEL
LIN {X 0,Y 460.567,Z 128.741,A -85,B 0,C 180,E1 -8119.616,E2 -8119.616} C_VEL
LIN {X 0,Y 460.512,Z 128.744,A -85,B 0,C 180,E1 -8122.429,E2 -8122.429} C_VEL
LIN {X 0,Y 460.536,Z 128.731,A -85,B 0,C 180,E1 -8125.793,E2 -8125.793} C_VEL
LIN {X 0,Y 460.521,Z 128.744,A -85,B 0,C 180,E1 -8129.232,E2 -8129.232} C_VEL
LIN {X 0,Y 460.526,Z 128.742,A -85,B 0,C 180,E1 -8132.285,E2 -8132.285} C_VEL
LIN {X 0,Y 460.506,Z 128.75,A -85,B 0,C 180,E1 -8135.446,E2 -8135.446} C_VEL
LIN {X 0,Y 460.495,Z 128.747,A -85,B 0,C 180,E1 -8138.89,E2 -8138.89} C_VEL
LIN {X 0,Y 460.503,Z 128.745,A -85,B 0,C 180,E1 -8141.598,E2 -8141.598} C_VEL
LIN {X 0,Y 460.512,Z 128.744,A -85,B 0,C 180,E1 -8144.589,E2 -8144.589} C_VEL
LIN {X 0,Y 460.475,Z 128.749,A -85,B 0,C 180,E1 -8147.813,E2 -8147.813} C_VEL
LIN {X 0,Y 460.51,Z 128.746,A -85,B 0,C 180,E1 -8150.135,E2 -8150.135} C_VEL
LIN {X 0,Y 460.46,Z 128.752,A -85,B 0,C 180,E1 -8153.469,E2 -8153.469} C_VEL
LIN {X 0,Y 460.501,Z 128.747,A -85,B 0,C 180,E1 -8156.673,E2 -8156.673} C_VEL
LIN {X 0,Y 460.478,Z 128.737,A -85,B 0,C 180,E1 -8159.758,E2 -8159.758} C_VEL
LIN {X 0,Y 460.527,Z 128.751,A -85,B 0,C 180,E1 -8162.594,E2 -8162.594} C_VEL
LIN {X 0,Y 463.798,Z 143.236,A -85,B 0,C 180,E1 -8165.394,E2 -8165.394} C_VEL
LIN {X 0,Y 464.004,Z 144.139,A -85,B 0,C 180,E1 -8165.534,E2 -8165.534} C_VEL
LIN {X 0,Y 466.227,Z 150.532,A -85,B 0,C 180,E1 -8165.765,E2 -8165.765} C_VEL
LIN {X 0,Y 469.497,Z 164.598,A -85,B 0,C 180,E1 -8166.178,E2 -8166.178} C_VEL
LIN {X 0,Y 468.741,Z 233.659,A -85,B 0,C 180,E1 -8167.267,E2 -8167.267} C_VEL
LIN {X 0,Y 467.969,Z 239.51,A -85,B 0,C 180,E1 -8167.322,E2 -8167.322} C_VEL
LIN {X 0,Y 462.495,Z 258.579,A -85,B 0,C 180,E1 -8167.351,E2 -8167.351} C_VEL
LIN {X 0,Y 461.801,Z 264.428,A -85,B 0,C 180,E1 -8167.411,E2 -8167.411} C_VEL
LIN {X 0,Y 461.186,Z 309.181,A -85,B 0,C 180,E1 -8168.142,E2 -8168.142} C_VEL
LIN {X 0,Y 460.703,Z 324.888,A -85,B 0,C 180,E1 -8168.576,E2 -8168.576} C_VEL
LIN {X 0,Y 460.155,Z 339.25,A -85,B 0,C 180,E1 -8169.15,E2 -8169.15} C_VEL
LIN {X 0,Y 459.328,Z 352.941,A -85,B 0,C 180,E1 -8169.863,E2 -8169.863} C_VEL
LIN {X 0,Y 458.482,Z 366.531,A -85,B 0,C 180,E1 -8170.757,E2 -8170.757} C_VEL
LIN {X 0,Y 457.565,Z 379.026,A -85,B 0,C 180,E1 -8171.763,E2 -8171.763} C_VEL
LIN {X 0,Y 456.707,Z 390.218,A -85,B 0,C 180,E1 -8172.842,E2 -8172.842} C_VEL
LIN {X 0,Y 455.829,Z 401.368,A -85,B 0,C 180,E1 -8174.117,E2 -8174.117} C_VEL
LIN {X 0,Y 455.043,Z 411.308,A -85,B 0,C 180,E1 -8175.465,E2 -8175.465} C_VEL
LIN {X 0,Y 454.272,Z 420.674,A -85,B 0,C 180,E1 -8176.973,E2 -8176.973} C_VEL
LIN {X 0,Y 453.767,Z 429.098,A -85,B 0,C 180,E1 -8178.611,E2 -8178.611} C_VEL
LIN {X 0,Y 453.253,Z 435.77,A -85,B 0,C 180,E1 -8180.179,E2 -8180.179} C_VEL
LIN {X 0,Y 452.916,Z 441.947,A -85,B 0,C 180,E1 -8181.972,E2 -8181.972} C_VEL
LIN {X 0,Y 452.731,Z 446.717,A -85,B 0,C 180,E1 -8183.762,E2 -8183.762} C_VEL
LIN {X 0,Y 452.514,Z 450.216,A -85,B 0,C 180,E1 -8185.546,E2 -8185.546} C_VEL
LIN {X 0,Y 452.525,Z 452.527,A -85,B 0,C 180,E1 -8187.33,E2 -8187.33} C_VEL
LIN {X 0,Y 452.428,Z 453.712,A -85,B 0,C 180,E1 -8189.11,E2 -8189.11} C_VEL
LIN {X 0,Y 452.428,Z 453.73,A -85,B 0,C 180,E1 -8190.89,E2 -8190.89} C_VEL
LIN {X 0,Y 452.525,Z 452.613,A -85,B 0,C 180,E1 -8192.671,E2 -8192.671} C_VEL
LIN {X 0,Y 452.512,Z 450.369,A -85,B 0,C 180,E1 -8194.454,E2 -8194.454} C_VEL
LIN {X 0,Y 452.73,Z 446.933,A -85,B 0,C 180,E1 -8196.238,E2 -8196.238} C_VEL
LIN {X 0,Y 452.914,Z 442.233,A -85,B 0,C 180,E1 -8198.028,E2 -8198.028} C_VEL
LIN {X 0,Y 453.235,Z 436.141,A -85,B 0,C 180,E1 -8199.821,E2 -8199.821} C_VEL
LIN {X 0,Y 453.81,Z 428.466,A -85,B 0,C 180,E1 -8201.615,E2 -8201.615} C_VEL
LIN {X 0,Y 454.311,Z 420.542,A -85,B 0,C 180,E1 -8203.143,E2 -8203.143} C_VEL
LIN {X 0,Y 455.08,Z 410.426,A -85,B 0,C 180,E1 -8204.763,E2 -8204.763} C_VEL
LIN {X 0,Y 455.887,Z 400.314,A -85,B 0,C 180,E1 -8206.111,E2 -8206.111} C_VEL
LIN {X 0,Y 456.793,Z 389.238,A -85,B 0,C 180,E1 -8207.354,E2 -8207.354} C_VEL
LIN {X 0,Y 457.646,Z 377.484,A -85,B 0,C 180,E1 -8208.466,E2 -8208.466} C_VEL
LIN {X 0,Y 458.622,Z 364.65,A -85,B 0,C 180,E1 -8209.469,E2 -8209.469} C_VEL
LIN {X 0,Y 459.518,Z 350.572,A -85,B 0,C 180,E1 -8210.362,E2 -8210.362} C_VEL
LIN {X 0,Y 460.272,Z 335.792,A -85,B 0,C 180,E1 -8211.094,E2 -8211.094} C_VEL
LIN {X 0,Y 460.847,Z 320.752,A -85,B 0,C 180,E1 -8211.646,E2 -8211.646} C_VEL
LIN {X 0,Y 461.279,Z 306.188,A -85,B 0,C 180,E1 -8212.006,E2 -8212.006} C_VEL
LIN {X 0,Y 463.057,Z 165.986,A -85,B 0,C 180,E1 -8214.25,E2 -8214.25} C_VEL
LIN {X 0,Y 459.227,Z 150.056,A -85,B 0,C 180,E1 -8214.736,E2 -8214.736} C_VEL
LIN {X 0,Y 456.78,Z 144.019,A -85,B 0,C 180,E1 -8215.002,E2 -8215.002} C_VEL
LIN {X 0,Y 453.613,Z 130.35,A -85,B 0,C 180,E1 -8217.698,E2 -8217.698} C_VEL
LIN {X 0,Y 453.486,Z 129.627,A -85,B 0,C 180,E1 -8217.854,E2 -8217.854} C_VEL
LIN {X 0,Y 453.447,Z 129.628,A -85,B 0,C 180,E1 -8220.762,E2 -8220.762} C_VEL
LIN {X 0,Y 453.454,Z 129.625,A -85,B 0,C 180,E1 -8223.915,E2 -8223.915} C_VEL
LIN {X 0,Y 453.432,Z 129.63,A -85,B 0,C 180,E1 -8227.192,E2 -8227.192} C_VEL
LIN {X 0,Y 453.464,Z 129.621,A -85,B 0,C 180,E1 -8230.612,E2 -8230.612} C_VEL
LIN {X 0,Y 453.481,Z 129.622,A -85,B 0,C 180,E1 -8234.528,E2 -8234.528} C_VEL
LIN {X 0,Y 453.443,Z 129.617,A -85,B 0,C 180,E1 -8238.205,E2 -8238.205} C_VEL
LIN {X 0,Y 453.44,Z 129.627,A -85,B 0,C 180,E1 -8240.802,E2 -8240.802} C_VEL
LIN {X 0,Y 453.444,Z 129.619,A -85,B 0,C 180,E1 -8243.916,E2 -8243.916} C_VEL
LIN {X 0,Y 453.474,Z 129.616,A -85,B 0,C 180,E1 -8247.15,E2 -8247.15} C_VEL
LIN {X 0,Y 453.449,Z 129.618,A -85,B 0,C 180,E1 -8250.266,E2 -8250.266} C_VEL
LIN {X 0,Y 453.443,Z 129.622,A -85,B 0,C 180,E1 -8253.29,E2 -8253.29} C_VEL
LIN {X 0,Y 453.494,Z 129.624,A -85,B 0,C 180,E1 -8256.238,E2 -8256.238} C_VEL
LIN {X 0,Y 453.476,Z 129.62,A -85,B 0,C 180,E1 -8259.117,E2 -8259.117} C_VEL
LIN {X 0,Y 453.488,Z 129.619,A -85,B 0,C 180,E1 -8261.943,E2 -8261.943} C_VEL
LIN {X 0,Y 453.523,Z 129.614,A -85,B 0,C 180,E1 -8264.726,E2 -8264.726} C_VEL
LIN {X 0,Y 453.561,Z 129.612,A -85,B 0,C 180,E1 -8268.379,E2 -8268.379} C_VEL
LIN {X 0,Y 453.58,Z 129.602,A -85,B 0,C 180,E1 -8271.086,E2 -8271.086} C_VEL
LIN {X 0,Y 453.639,Z 129.605,A -85,B 0,C 180,E1 -8273.774,E2 -8273.774} C_VEL
LIN {X 0,Y 453.707,Z 129.593,A -85,B 0,C 180,E1 -8277.336,E2 -8277.336} C_VEL
LIN {X 0,Y 453.794,Z 129.579,A -85,B 0,C 180,E1 -8280,E2 -8280} C_VEL
LIN {X 0,Y 453.736,Z 129.587,A -85,B 0,C 180,E1 -8282.663,E2 -8282.663} C_VEL
LIN {X 0,Y 453.647,Z 129.599,A -85,B 0,C 180,E1 -8286.226,E2 -8286.226} C_VEL
LIN {X 0,Y 453.587,Z 129.607,A -85,B 0,C 180,E1 -8288.913,E2 -8288.913} C_VEL
LIN {X 0,Y 453.567,Z 129.609,A -85,B 0,C 180,E1 -8292.529,E2 -8292.529} C_VEL
LIN {X 0,Y 453.547,Z 129.612,A -85,B 0,C 180,E1 -8296.196,E2 -8296.196} C_VEL
LIN {X 0,Y 453.519,Z 129.617,A -85,B 0,C 180,E1 -8299.039,E2 -8299.039} C_VEL
LIN {X 0,Y 453.479,Z 129.617,A -85,B 0,C 180,E1 -8301.836,E2 -8301.836} C_VEL
LIN {X 0,Y 453.496,Z 129.624,A -85,B 0,C 180,E1 -8304.735,E2 -8304.735} C_VEL
LIN {X 0,Y 453.508,Z 129.616,A -85,B 0,C 180,E1 -8307.953,E2 -8307.953} C_VEL
LIN {X 0,Y 453.477,Z 129.626,A -85,B 0,C 180,E1 -8310.759,E2 -8310.759} C_VEL
LIN {X 0,Y 453.47,Z 129.617,A -85,B 0,C 180,E1 -8313.913,E2 -8313.913} C_VEL
LIN {X 0,Y 453.454,Z 129.622,A -85,B 0,C 180,E1 -8317.189,E2 -8317.189} C_VEL
LIN {X 0,Y 453.485,Z 129.617,A -85,B 0,C 180,E1 -8319.45,E2 -8319.45} C_VEL
LIN {X 0,Y 453.478,Z 129.622,A -85,B 0,C 180,E1 -8321.935,E2 -8321.935} C_VEL
LIN {X 0,Y 453.486,Z 129.619,A -85,B 0,C 180,E1 -8325.471,E2 -8325.471} C_VEL
LIN {X 0,Y 453.481,Z 129.624,A -85,B 0,C 180,E1 -8328.209,E2 -8328.209} C_VEL
LIN {X 0,Y 453.511,Z 129.617,A -85,B 0,C 180,E1 -8330.791,E2 -8330.791} C_VEL
LIN {X 0,Y 453.455,Z 129.626,A -85,B 0,C 180,E1 -8333.917,E2 -8333.917} C_VEL
LIN {X 0,Y 453.484,Z 129.622,A -85,B 0,C 180,E1 -8337.151,E2 -8337.151} C_VEL
LIN {X 0,Y 453.502,Z 129.673,A -85,B 0,C 180,E1 -8338.935,E2 -8338.935} C_VEL
LIN {X 0,Y 457.481,Z 145.785,A -85,B 0,C 180,E1 -8341.81,E2 -8341.81} C_VEL
LIN {X 0,Y 458.548,Z 151.26,A -85,B 0,C 180,E1 -8342.741,E2 -8342.741} C_VEL
LIN {X 0,Y 457.617,Z 166.667,A -85,B 0,C 180,E1 -8345.1,E2 -8345.1} C_VEL
LIN {X 0,Y 462.799,Z 193.148,A -85,B 0,C 180,E1 -8345.84,E2 -8345.84} C_VEL
LIN {X 0,Y 461.237,Z 317.518,A -85,B 0,C 180,E1 -8347.815,E2 -8347.815} C_VEL
LIN {X 0,Y 460.857,Z 337.091,A -85,B 0,C 180,E1 -8348.178,E2 -8348.178} C_VEL
LIN {X 0,Y 460.216,Z 352.32,A -85,B 0,C 180,E1 -8348.636,E2 -8348.636} C_VEL
LIN {X 0,Y 459.51,Z 367.237,A -85,B 0,C 180,E1 -8349.272,E2 -8349.272} C_VEL
LIN {X 0,Y 458.576,Z 381.488,A -85,B 0,C 180,E1 -8350.062,E2 -8350.062} C_VEL
LIN {X 0,Y 457.673,Z 394.358,A -85,B 0,C 180,E1 -8350.955,E2 -8350.955} C_VEL
LIN {X 0,Y 456.673,Z 407.561,A -85,B 0,C 180,E1 -8352.074,E2 -8352.074} C_VEL
LIN {X 0,Y 455.901,Z 418.641,A -85,B 0,C 180,E1 -8353.199,E2 -8353.199} C_VEL
LIN {X 0,Y 454.925,Z 429.832,A -85,B 0,C 180,E1 -8354.544,E2 -8354.544} C_VEL
LIN {X 0,Y 454.148,Z 440.697,A -85,B 0,C 180,E1 -8356.121,E2 -8356.121} C_VEL
LIN {X 0,Y 453.556,Z 449.462,A -85,B 0,C 180,E1 -8357.643,E2 -8357.643} C_VEL
LIN {X 0,Y 453.169,Z 457.259,A -85,B 0,C 180,E1 -8359.274,E2 -8359.274} C_VEL
LIN {X 0,Y 452.781,Z 464.266,A -85,B 0,C 180,E1 -8361.07,E2 -8361.07} C_VEL
LIN {X 0,Y 452.645,Z 469.779,A -85,B 0,C 180,E1 -8362.865,E2 -8362.865} C_VEL
LIN {X 0,Y 452.509,Z 473.946,A -85,B 0,C 180,E1 -8364.653,E2 -8364.653} C_VEL
LIN {X 0,Y 452.427,Z 476.867,A -85,B 0,C 180,E1 -8366.438,E2 -8366.438} C_VEL
LIN {X 0,Y 452.433,Z 478.611,A -85,B 0,C 180,E1 -8368.22,E2 -8368.22} C_VEL
LIN {X 0,Y 452.432,Z 479.208,A -85,B 0,C 180,E1 -8370,E2 -8370} C_VEL
LIN {X 0,Y 452.433,Z 478.607,A -85,B 0,C 180,E1 -8371.78,E2 -8371.78} C_VEL
LIN {X 0,Y 452.427,Z 476.86,A -85,B 0,C 180,E1 -8373.562,E2 -8373.562} C_VEL
LIN {X 0,Y 452.513,Z 473.941,A -85,B 0,C 180,E1 -8375.347,E2 -8375.347} C_VEL
LIN {X 0,Y 452.645,Z 469.778,A -85,B 0,C 180,E1 -8377.135,E2 -8377.135} C_VEL
LIN {X 0,Y 452.781,Z 464.26,A -85,B 0,C 180,E1 -8378.929,E2 -8378.929} C_VEL
LIN {X 0,Y 453.166,Z 457.243,A -85,B 0,C 180,E1 -8380.726,E2 -8380.726} C_VEL
LIN {X 0,Y 453.564,Z 448.509,A -85,B 0,C 180,E1 -8382.529,E2 -8382.529} C_VEL
LIN {X 0,Y 454.273,Z 439.238,A -85,B 0,C 180,E1 -8384.103,E2 -8384.103} C_VEL
LIN {X 0,Y 454.922,Z 429.812,A -85,B 0,C 180,E1 -8385.456,E2 -8385.456} C_VEL
LIN {X 0,Y 455.937,Z 417.597,A -85,B 0,C 180,E1 -8386.915,E2 -8386.915} C_VEL
LIN {X 0,Y 456.855,Z 405.14,A -85,B 0,C 180,E1 -8388.151,E2 -8388.151} C_VEL
LIN {X 0,Y 457.902,Z 391.364,A -85,B 0,C 180,E1 -8389.268,E2 -8389.268} C_VEL
LIN {X 0,Y 458.851,Z 377.839,A -85,B 0,C 180,E1 -8390.159,E2 -8390.159} C_VEL
LIN {X 0,Y 459.767,Z 363.09,A -85,B 0,C 180,E1 -8390.923,E2 -8390.923} C_VEL
LIN {X 0,Y 460.424,Z 348.694,A -85,B 0,C 180,E1 -8391.49,E2 -8391.49} C_VEL
LIN {X 0,Y 460.945,Z 333.529,A -85,B 0,C 180,E1 -8391.905,E2 -8391.905} C_VEL
LIN {X 0,Y 462.62,Z 213.306,A -85,B 0,C 180,E1 -8393.831,E2 -8393.831} C_VEL
LIN {X 0,Y 462.688,Z 192.521,A -85,B 0,C 180,E1 -8394.173,E2 -8394.173} C_VEL
LIN {X 0,Y 457.611,Z 166.584,A -85,B 0,C 180,E1 -8394.908,E2 -8394.908} C_VEL
LIN {X 0,Y 458.54,Z 151.231,A -85,B 0,C 180,E1 -8397.257,E2 -8397.257} C_VEL
LIN {X 0,Y 456.332,Z 140.889,A -85,B 0,C 180,E1 -8399.04,E2 -8399.04} C_VEL
LIN {X 0,Y 453.492,Z 129.619,A -85,B 0,C 180,E1 -8401.096,E2 -8401.096} C_VEL
LIN {X 0,Y 453.477,Z 129.621,A -85,B 0,C 180,E1 -8403.913,E2 -8403.913} C_VEL
LIN {X 0,Y 453.453,Z 129.625,A -85,B 0,C 180,E1 -8407.19,E2 -8407.19} C_VEL
LIN {X 0,Y 453.518,Z 129.618,A -85,B 0,C 180,E1 -8409.447,E2 -8409.447} C_VEL
LIN {X 0,Y 453.463,Z 129.621,A -85,B 0,C 180,E1 -8412.995,E2 -8412.995} C_VEL
LIN {X 0,Y 453.465,Z 129.626,A -85,B 0,C 180,E1 -8415.779,E2 -8415.779} C_VEL
LIN {X 0,Y 453.48,Z 129.62,A -85,B 0,C 180,E1 -8418.209,E2 -8418.209} C_VEL
LIN {X 0,Y 453.488,Z 129.618,A -85,B 0,C 180,E1 -8420.795,E2 -8420.795} C_VEL
LIN {X 0,Y 453.455,Z 129.621,A -85,B 0,C 180,E1 -8423.917,E2 -8423.917} C_VEL
LIN {X 0,Y 453.48,Z 129.621,A -85,B 0,C 180,E1 -8427.151,E2 -8427.151} C_VEL
LIN {X 0,Y 453.475,Z 129.617,A -85,B 0,C 180,E1 -8430.268,E2 -8430.268} C_VEL
LIN {X 0,Y 453.533,Z 129.612,A -85,B 0,C 180,E1 -8432.297,E2 -8432.297} C_VEL
LIN {X 0,Y 453.493,Z 129.621,A -85,B 0,C 180,E1 -8435.264,E2 -8435.264} C_VEL
LIN {X 0,Y 453.482,Z 129.62,A -85,B 0,C 180,E1 -8438.415,E2 -8438.415} C_VEL
LIN {X 0,Y 453.524,Z 129.619,A -85,B 0,C 180,E1 -8441.009,E2 -8441.009} C_VEL
LIN {X 0,Y 453.571,Z 129.604,A -85,B 0,C 180,E1 -8443.88,E2 -8443.88} C_VEL
LIN {X 0,Y 453.566,Z 129.605,A -85,B 0,C 180,E1 -8447.471,E2 -8447.471} C_VEL
LIN {X 0,Y 453.586,Z 129.604,A -85,B 0,C 180,E1 -8451.087,E2 -8451.087} C_VEL
LIN {X 0,Y 453.647,Z 129.599,A -85,B 0,C 180,E1 -8453.774,E2 -8453.774} C_VEL
LIN {X 0,Y 453.737,Z 129.587,A -85,B 0,C 180,E1 -8457.337,E2 -8457.337} C_VEL
LIN {X 0,Y 453.794,Z 129.581,A -85,B 0,C 180,E1 -8460,E2 -8460} C_VEL
LIN {X 0,Y 453.708,Z 129.594,A -85,B 0,C 180,E1 -8462.664,E2 -8462.664} C_VEL
LIN {X 0,Y 453.644,Z 129.604,A -85,B 0,C 180,E1 -8466.226,E2 -8466.226} C_VEL
LIN {X 0,Y 453.58,Z 129.603,A -85,B 0,C 180,E1 -8468.914,E2 -8468.914} C_VEL
LIN {X 0,Y 453.567,Z 129.606,A -85,B 0,C 180,E1 -8472.529,E2 -8472.529} C_VEL
LIN {X 0,Y 453.505,Z 129.619,A -85,B 0,C 180,E1 -8476.091,E2 -8476.091} C_VEL
LIN {X 0,Y 453.519,Z 129.615,A -85,B 0,C 180,E1 -8479.039,E2 -8479.039} C_VEL
LIN {X 0,Y 453.478,Z 129.623,A -85,B 0,C 180,E1 -8481.836,E2 -8481.836} C_VEL
LIN {X 0,Y 453.471,Z 129.617,A -85,B 0,C 180,E1 -8484.737,E2 -8484.737} C_VEL
LIN {X 0,Y 453.464,Z 129.621,A -85,B 0,C 180,E1 -8487.943,E2 -8487.943} C_VEL
LIN {X 0,Y 453.458,Z 129.622,A -85,B 0,C 180,E1 -8490.761,E2 -8490.761} C_VEL
LIN {X 0,Y 453.467,Z 129.62,A -85,B 0,C 180,E1 -8493.914,E2 -8493.914} C_VEL
LIN {X 0,Y 453.447,Z 129.626,A -85,B 0,C 180,E1 -8497.19,E2 -8497.19} C_VEL
LIN {X 0,Y 453.471,Z 129.619,A -85,B 0,C 180,E1 -8500.612,E2 -8500.612} C_VEL
LIN {X 0,Y 453.482,Z 129.619,A -85,B 0,C 180,E1 -8504.528,E2 -8504.528} C_VEL
LIN {X 0,Y 453.437,Z 129.626,A -85,B 0,C 180,E1 -8508.071,E2 -8508.071} C_VEL
LIN {X 0,Y 453.439,Z 129.626,A -85,B 0,C 180,E1 -8510.802,E2 -8510.802} C_VEL
LIN {X 0,Y 453.442,Z 129.624,A -85,B 0,C 180,E1 -8513.916,E2 -8513.916} C_VEL
LIN {X 0,Y 453.465,Z 129.623,A -85,B 0,C 180,E1 -8516.816,E2 -8516.816} C_VEL
LIN {X 0,Y 453.447,Z 129.611,A -85,B 0,C 180,E1 -8520.266,E2 -8520.266} C_VEL
LIN {X 0,Y 453.505,Z 129.821,A -85,B 0,C 180,E1 -8522.295,E2 -8522.295} C_VEL
LIN {X 0,Y 456.702,Z 143.706,A -85,B 0,C 180,E1 -8525.031,E2 -8525.031} C_VEL
LIN {X 0,Y 456.876,Z 144.478,A -85,B 0,C 180,E1 -8525.128,E2 -8525.128} C_VEL
LIN {X 0,Y 459.992,Z 152.722,A -85,B 0,C 180,E1 -8525.449,E2 -8525.449} C_VEL
LIN {X 0,Y 463.098,Z 166.798,A -85,B 0,C 180,E1 -8525.861,E2 -8525.861} C_VEL
LIN {X 0,Y 461.801,Z 264.428,A -85,B 0,C 180,E1 -8527.411,E2 -8527.411} C_VEL
LIN {X 0,Y 461.08,Z 270.277,A -85,B 0,C 180,E1 -8527.47,E2 -8527.47} C_VEL
LIN {X 0,Y 455.532,Z 289.323,A -85,B 0,C 180,E1 -8527.497,E2 -8527.497} C_VEL
LIN {X 0,Y 454.88,Z 295.169,A -85,B 0,C 180,E1 -8527.56,E2 -8527.56} C_VEL
LIN {X 0,Y 454.448,Z 313.81,A -85,B 0,C 180,E1 -8527.916,E2 -8527.916} C_VEL
LIN {X 0,Y 453.946,Z 329.163,A -85,B 0,C 180,E1 -8528.4,E2 -8528.4} C_VEL
LIN {X 0,Y 453.328,Z 343.217,A -85,B 0,C 180,E1 -8529.018,E2 -8529.018} C_VEL
LIN {X 0,Y 452.488,Z 356.797,A -85,B 0,C 180,E1 -8529.782,E2 -8529.782} C_VEL
LIN {X 0,Y 451.551,Z 369.729,A -85,B 0,C 180,E1 -8530.686,E2 -8530.686} C_VEL
LIN {X 0,Y 450.626,Z 381.77,A -85,B 0,C 180,E1 -8531.707,E2 -8531.707} C_VEL
LIN {X 0,Y 449.583,Z 393.987,A -85,B 0,C 180,E1 -8532.956,E2 -8532.956} C_VEL
LIN {X 0,Y 448.689,Z 405.11,A -85,B 0,C 180,E1 -8534.324,E2 -8534.324} C_VEL
LIN {X 0,Y 447.729,Z 415.916,A -85,B 0,C 180,E1 -8535.918,E2 -8535.918} C_VEL
LIN {X 0,Y 447.027,Z 424.877,A -85,B 0,C 180,E1 -8537.516,E2 -8537.516} C_VEL
LIN {X 0,Y 446.445,Z 432.304,A -85,B 0,C 180,E1 -8539.111,E2 -8539.111} C_VEL
LIN {X 0,Y 446.016,Z 439.245,A -85,B 0,C 180,E1 -8540.934,E2 -8540.934} C_VEL
LIN {X 0,Y 445.722,Z 444.7,A -85,B 0,C 180,E1 -8542.753,E2 -8542.753} C_VEL
LIN {X 0,Y 445.581,Z 448.817,A -85,B 0,C 180,E1 -8544.57,E2 -8544.57} C_VEL
LIN {X 0,Y 445.441,Z 451.714,A -85,B 0,C 180,E1 -8546.382,E2 -8546.382} C_VEL
LIN {X 0,Y 445.376,Z 453.458,A -85,B 0,C 180,E1 -8548.191,E2 -8548.191} C_VEL
LIN {X 0,Y 445.342,Z 454.069,A -85,B 0,C 180,E1 -8550,E2 -8550} C_VEL
LIN {X 0,Y 445.377,Z 453.509,A -85,B 0,C 180,E1 -8551.809,E2 -8551.809} C_VEL
LIN {X 0,Y 445.441,Z 451.833,A -85,B 0,C 180,E1 -8553.618,E2 -8553.618} C_VEL
LIN {X 0,Y 445.574,Z 449.001,A -85,B 0,C 180,E1 -8555.431,E2 -8555.431} C_VEL
LIN {X 0,Y 445.714,Z 444.947,A -85,B 0,C 180,E1 -8557.247,E2 -8557.247} C_VEL
LIN {X 0,Y 446.005,Z 439.569,A -85,B 0,C 180,E1 -8559.066,E2 -8559.066} C_VEL
LIN {X 0,Y 446.431,Z 432.716,A -85,B 0,C 180,E1 -8560.889,E2 -8560.889} C_VEL
LIN {X 0,Y 446.992,Z 425.341,A -85,B 0,C 180,E1 -8562.485,E2 -8562.485} C_VEL
LIN {X 0,Y 447.689,Z 416.457,A -85,B 0,C 180,E1 -8564.083,E2 -8564.083} C_VEL
LIN {X 0,Y 448.434,Z 407.397,A -85,B 0,C 180,E1 -8565.452,E2 -8565.452} C_VEL
LIN {X 0,Y 449.353,Z 396.706,A -85,B 0,C 180,E1 -8566.819,E2 -8566.819} C_VEL
LIN {X 0,Y 450.359,Z 385.037,A -85,B 0,C 180,E1 -8568.068,E2 -8568.068} C_VEL
LIN {X 0,Y 451.358,Z 372.281,A -85,B 0,C 180,E1 -8569.204,E2 -8569.204} C_VEL
LIN {X 0,Y 452.358,Z 358.206,A -85,B 0,C 180,E1 -8570.224,E2 -8570.224} C_VEL
LIN {X 0,Y 453.317,Z 343.479,A -85,B 0,C 180,E1 -8571.063,E2 -8571.063} C_VEL
LIN {X 0,Y 453.998,Z 328.548,A -85,B 0,C 180,E1 -8571.715,E2 -8571.715} C_VEL
LIN {X 0,Y 454.53,Z 312.778,A -85,B 0,C 180,E1 -8572.201,E2 -8572.201} C_VEL
LIN {X 0,Y 454.913,Z 292.928,A -85,B 0,C 180,E1 -8572.57,E2 -8572.57} C_VEL
LIN {X 0,Y 456.588,Z 167.159,A -85,B 0,C 180,E1 -8574.599,E2 -8574.599} C_VEL
LIN {X 0,Y 453.094,Z 152.815,A -85,B 0,C 180,E1 -8575.049,E2 -8575.049} C_VEL
LIN {X 0,Y 449.62,Z 144.259,A -85,B 0,C 180,E1 -8575.422,E2 -8575.422} C_VEL
LIN {X 0,Y 446.416,Z 130.539,A -85,B 0,C 180,E1 -8578.184,E2 -8578.184} C_VEL
LIN {X 0,Y 446.389,Z 130.509,A -85,B 0,C 180,E1 -8581.303,E2 -8581.303} C_VEL
LIN {X 0,Y 446.412,Z 130.502,A -85,B 0,C 180,E1 -8584.525,E2 -8584.525} C_VEL
LIN {X 0,Y 446.387,Z 130.508,A -85,B 0,C 180,E1 -8587.881,E2 -8587.881} C_VEL
LIN {X 0,Y 446.395,Z 130.507,A -85,B 0,C 180,E1 -8591.395,E2 -8591.395} C_VEL
LIN {X 0,Y 446.419,Z 130.505,A -85,B 0,C 180,E1 -8595.108,E2 -8595.108} C_VEL
LIN {X 0,Y 446.401,Z 130.498,A -85,B 0,C 180,E1 -8598.606,E2 -8598.606} C_VEL
LIN {X 0,Y 446.399,Z 130.497,A -85,B 0,C 180,E1 -8601.924,E2 -8601.924} C_VEL
LIN {X 0,Y 446.421,Z 130.499,A -85,B 0,C 180,E1 -8605.476,E2 -8605.476} C_VEL
LIN {X 0,Y 446.392,Z 130.492,A -85,B 0,C 180,E1 -8608.698,E2 -8608.698} C_VEL
LIN {X 0,Y 446.403,Z 130.502,A -85,B 0,C 180,E1 -8611.842,E2 -8611.842} C_VEL
LIN {X 0,Y 446.423,Z 130.501,A -85,B 0,C 180,E1 -8614.846,E2 -8614.846} C_VEL
LIN {X 0,Y 446.449,Z 130.497,A -85,B 0,C 180,E1 -8618.246,E2 -8618.246} C_VEL
LIN {X 0,Y 446.442,Z 130.496,A -85,B 0,C 180,E1 -8621.648,E2 -8621.648} C_VEL
LIN {X 0,Y 446.463,Z 130.495,A -85,B 0,C 180,E1 -8624.478,E2 -8624.478} C_VEL
LIN {X 0,Y 446.519,Z 130.485,A -85,B 0,C 180,E1 -8627.384,E2 -8627.384} C_VEL
LIN {X 0,Y 446.528,Z 130.479,A -85,B 0,C 180,E1 -8630.944,E2 -8630.944} C_VEL
LIN {X 0,Y 446.609,Z 130.481,A -85,B 0,C 180,E1 -8633.676,E2 -8633.676} C_VEL
LIN {X 0,Y 446.656,Z 130.471,A -85,B 0,C 180,E1 -8637.294,E2 -8637.294} C_VEL
LIN {X 0,Y 446.764,Z 130.455,A -85,B 0,C 180,E1 -8640,E2 -8640} C_VEL
LIN {X 0,Y 446.683,Z 130.466,A -85,B 0,C 180,E1 -8642.705,E2 -8642.705} C_VEL
LIN {X 0,Y 446.616,Z 130.475,A -85,B 0,C 180,E1 -8646.324,E2 -8646.324} C_VEL
LIN {X 0,Y 446.534,Z 130.486,A -85,B 0,C 180,E1 -8649.055,E2 -8649.055} C_VEL
LIN {X 0,Y 446.524,Z 130.488,A -85,B 0,C 180,E1 -8652.73,E2 -8652.73} C_VEL
LIN {X 0,Y 446.491,Z 130.492,A -85,B 0,C 180,E1 -8656.459,E2 -8656.459} C_VEL
LIN {X 0,Y 446.471,Z 130.499,A -85,B 0,C 180,E1 -8659.303,E2 -8659.303} C_VEL
LIN {X 0,Y 446.42,Z 130.497,A -85,B 0,C 180,E1 -8662.199,E2 -8662.199} C_VEL
LIN {X 0,Y 446.44,Z 130.499,A -85,B 0,C 180,E1 -8665.153,E2 -8665.153} C_VEL
LIN {X 0,Y 446.451,Z 130.496,A -85,B 0,C 180,E1 -8668.181,E2 -8668.181} C_VEL
LIN {X 0,Y 446.417,Z 130.501,A -85,B 0,C 180,E1 -8671.3,E2 -8671.3} C_VEL
LIN {X 0,Y 446.424,Z 130.5,A -85,B 0,C 180,E1 -8674.523,E2 -8674.523} C_VEL
LIN {X 0,Y 446.415,Z 130.5,A -85,B 0,C 180,E1 -8678.079,E2 -8678.079} C_VEL
LIN {X 0,Y 446.428,Z 130.501,A -85,B 0,C 180,E1 -8680.917,E2 -8680.917} C_VEL
LIN {X 0,Y 446.401,Z 130.504,A -85,B 0,C 180,E1 -8683.846,E2 -8683.846} C_VEL
LIN {X 0,Y 446.399,Z 130.505,A -85,B 0,C 180,E1 -8686.403,E2 -8686.403} C_VEL
LIN {X 0,Y 446.428,Z 130.494,A -85,B 0,C 180,E1 -8689.082,E2 -8689.082} C_VEL
LIN {X 0,Y 446.417,Z 130.503,A -85,B 0,C 180,E1 -8691.92,E2 -8691.92} C_VEL
LIN {X 0,Y 446.43,Z 130.501,A -85,B 0,C 180,E1 -8695.477,E2 -8695.477} C_VEL
LIN {X 0,Y 446.443,Z 130.562,A -85,B 0,C 180,E1 -8698.571,E2 -8698.571} C_VEL
LIN {X 0,Y 450.097,Z 145.195,A -85,B 0,C 180,E1 -8701.244,E2 -8701.244} C_VEL
LIN {X 0,Y 451.666,Z 152.303,A -85,B 0,C 180,E1 -8702.49,E2 -8702.49} C_VEL
LIN {X 0,Y 451.048,Z 163.997,A -85,B 0,C 180,E1 -8704.319,E2 -8704.319} C_VEL
LIN {X 0,Y 450.852,Z 166.525,A -85,B 0,C 180,E1 -8704.705,E2 -8704.705} C_VEL
LIN {X 0,Y 456.356,Z 194.728,A -85,B 0,C 180,E1 -8705.506,E2 -8705.506} C_VEL
LIN {X 0,Y 454.427,Z 332.163,A -85,B 0,C 180,E1 -8707.734,E2 -8707.734} C_VEL
LIN {X 0,Y 453.844,Z 347.722,A -85,B 0,C 180,E1 -8708.152,E2 -8708.152} C_VEL
LIN {X 0,Y 453.095,Z 362.09,A -85,B 0,C 180,E1 -8708.714,E2 -8708.714} C_VEL
LIN {X 0,Y 452.299,Z 375.718,A -85,B 0,C 180,E1 -8709.417,E2 -8709.417} C_VEL
LIN {X 0,Y 451.271,Z 389.628,A -85,B 0,C 180,E1 -8710.319,E2 -8710.319} C_VEL
LIN {X 0,Y 450.284,Z 402.376,A -85,B 0,C 180,E1 -8711.339,E2 -8711.339} C_VEL
LIN {X 0,Y 449.231,Z 415.489,A -85,B 0,C 180,E1 -8712.614,E2 -8712.614} C_VEL
LIN {X 0,Y 448.389,Z 426.072,A -85,B 0,C 180,E1 -8713.846,E2 -8713.846} C_VEL
LIN {X 0,Y 447.554,Z 436.066,A -85,B 0,C 180,E1 -8715.216,E2 -8715.216} C_VEL
LIN {X 0,Y 446.767,Z 445.846,A -85,B 0,C 180,E1 -8716.815,E2 -8716.815} C_VEL
LIN {X 0,Y 446.288,Z 454.012,A -85,B 0,C 180,E1 -8718.417,E2 -8718.417} C_VEL
LIN {X 0,Y 445.825,Z 460.76,A -85,B 0,C 180,E1 -8720.014,E2 -8720.014} C_VEL
LIN {X 0,Y 445.606,Z 466.999,A -85,B 0,C 180,E1 -8721.839,E2 -8721.839} C_VEL
LIN {X 0,Y 445.451,Z 471.926,A -85,B 0,C 180,E1 -8723.703,E2 -8723.703} C_VEL
LIN {X 0,Y 445.36,Z 475.358,A -85,B 0,C 180,E1 -8725.474,E2 -8725.474} C_VEL
LIN {X 0,Y 445.418,Z 477.687,A -85,B 0,C 180,E1 -8727.287,E2 -8727.287} C_VEL
LIN {X 0,Y 445.335,Z 478.855,A -85,B 0,C 180,E1 -8729.096,E2 -8729.096} C_VEL
LIN {X 0,Y 445.335,Z 478.854,A -85,B 0,C 180,E1 -8730.904,E2 -8730.904} C_VEL
LIN {X 0,Y 445.418,Z 477.681,A -85,B 0,C 180,E1 -8732.713,E2 -8732.713} C_VEL
LIN {X 0,Y 445.361,Z 475.35,A -85,B 0,C 180,E1 -8734.525,E2 -8734.525} C_VEL
LIN {X 0,Y 445.488,Z 471.82,A -85,B 0,C 180,E1 -8736.34,E2 -8736.34} C_VEL
LIN {X 0,Y 445.606,Z 466.995,A -85,B 0,C 180,E1 -8738.16,E2 -8738.16} C_VEL
LIN {X 0,Y 445.824,Z 460.747,A -85,B 0,C 180,E1 -8739.986,E2 -8739.986} C_VEL
LIN {X 0,Y 446.256,Z 453.993,A -85,B 0,C 180,E1 -8741.584,E2 -8741.584} C_VEL
LIN {X 0,Y 446.766,Z 445.829,A -85,B 0,C 180,E1 -8743.185,E2 -8743.185} C_VEL
LIN {X 0,Y 447.554,Z 436.047,A -85,B 0,C 180,E1 -8744.784,E2 -8744.784} C_VEL
LIN {X 0,Y 448.336,Z 426.046,A -85,B 0,C 180,E1 -8746.155,E2 -8746.155} C_VEL
LIN {X 0,Y 449.314,Z 414.389,A -85,B 0,C 180,E1 -8747.5,E2 -8747.5} C_VEL
LIN {X 0,Y 450.244,Z 402.342,A -85,B 0,C 180,E1 -8748.662,E2 -8748.662} C_VEL
LIN {X 0,Y 451.262,Z 389.572,A -85,B 0,C 180,E1 -8749.681,E2 -8749.681} C_VEL
LIN {X 0,Y 452.282,Z 375.644,A -85,B 0,C 180,E1 -8750.583,E2 -8750.583} C_VEL
LIN {X 0,Y 453.179,Z 361.578,A -85,B 0,C 180,E1 -8751.302,E2 -8751.302} C_VEL
LIN {X 0,Y 453.865,Z 346.693,A -85,B 0,C 180,E1 -8751.876,E2 -8751.876} C_VEL
LIN {X 0,Y 454.403,Z 331.949,A -85,B 0,C 180,E1 -8752.267,E2 -8752.267} C_VEL
LIN {X 0,Y 456.352,Z 197.314,A -85,B 0,C 180,E1 -8754.445,E2 -8754.445} C_VEL
LIN {X 0,Y 456.054,Z 192.918,A -85,B 0,C 180,E1 -8754.537,E2 -8754.537} C_VEL
LIN {X 0,Y 450.861,Z 166.437,A -85,B 0,C 180,E1 -8755.298,E2 -8755.298} C_VEL
LIN {X 0,Y 451.74,Z 153.417,A -85,B 0,C 180,E1 -8757.32,E2 -8757.32} C_VEL
LIN {X 0,Y 450.09,Z 145.166,A -85,B 0,C 180,E1 -8758.755,E2 -8758.755} C_VEL
LIN {X 0,Y 446.437,Z 130.498,A -85,B 0,C 180,E1 -8761.452,E2 -8761.452} C_VEL
LIN {X 0,Y 446.429,Z 130.498,A -85,B 0,C 180,E1 -8764.523,E2 -8764.523} C_VEL
LIN {X 0,Y 446.416,Z 130.505,A -85,B 0,C 180,E1 -8768.079,E2 -8768.079} C_VEL
LIN {X 0,Y 446.428,Z 130.498,A -85,B 0,C 180,E1 -8770.918,E2 -8770.918} C_VEL
LIN {X 0,Y 446.401,Z 130.506,A -85,B 0,C 180,E1 -8773.846,E2 -8773.846} C_VEL
LIN {X 0,Y 446.399,Z 130.501,A -85,B 0,C 180,E1 -8776.404,E2 -8776.404} C_VEL
LIN {X 0,Y 446.428,Z 130.499,A -85,B 0,C 180,E1 -8779.083,E2 -8779.083} C_VEL
LIN {X 0,Y 446.409,Z 130.5,A -85,B 0,C 180,E1 -8782.121,E2 -8782.121} C_VEL
LIN {X 0,Y 446.424,Z 130.502,A -85,B 0,C 180,E1 -8785.477,E2 -8785.477} C_VEL
LIN {X 0,Y 446.417,Z 130.499,A -85,B 0,C 180,E1 -8788.7,E2 -8788.7} C_VEL
LIN {X 0,Y 446.486,Z 130.491,A -85,B 0,C 180,E1 -8791.822,E2 -8791.822} C_VEL
LIN {X 0,Y 446.438,Z 130.5,A -85,B 0,C 180,E1 -8794.847,E2 -8794.847} C_VEL
LIN {X 0,Y 446.45,Z 130.496,A -85,B 0,C 180,E1 -8798.245,E2 -8798.245} C_VEL
LIN {X 0,Y 446.452,Z 130.496,A -85,B 0,C 180,E1 -8801.649,E2 -8801.649} C_VEL
LIN {X 0,Y 446.509,Z 130.487,A -85,B 0,C 180,E1 -8804.48,E2 -8804.48} C_VEL
LIN {X 0,Y 446.519,Z 130.484,A -85,B 0,C 180,E1 -8808.193,E2 -8808.193} C_VEL
LIN {X 0,Y 446.534,Z 130.484,A -85,B 0,C 180,E1 -8810.945,E2 -8810.945} C_VEL
LIN {X 0,Y 446.615,Z 130.475,A -85,B 0,C 180,E1 -8813.676,E2 -8813.676} C_VEL
LIN {X 0,Y 446.684,Z 130.466,A -85,B 0,C 180,E1 -8817.295,E2 -8817.295} C_VEL
LIN {X 0,Y 446.764,Z 130.457,A -85,B 0,C 180,E1 -8820,E2 -8820} C_VEL
LIN {X 0,Y 446.658,Z 130.471,A -85,B 0,C 180,E1 -8822.706,E2 -8822.706} C_VEL
LIN {X 0,Y 446.613,Z 130.481,A -85,B 0,C 180,E1 -8826.324,E2 -8826.324} C_VEL
LIN {X 0,Y 446.529,Z 130.481,A -85,B 0,C 180,E1 -8829.056,E2 -8829.056} C_VEL
LIN {X 0,Y 446.524,Z 130.482,A -85,B 0,C 180,E1 -8832.73,E2 -8832.73} C_VEL
LIN {X 0,Y 446.456,Z 130.495,A -85,B 0,C 180,E1 -8836.209,E2 -8836.209} C_VEL
LIN {X 0,Y 446.47,Z 130.494,A -85,B 0,C 180,E1 -8839.303,E2 -8839.303} C_VEL
LIN {X 0,Y 446.42,Z 130.502,A -85,B 0,C 180,E1 -8842.2,E2 -8842.2} C_VEL
LIN {X 0,Y 446.423,Z 130.496,A -85,B 0,C 180,E1 -8845.154,E2 -8845.154} C_VEL
LIN {X 0,Y 446.438,Z 130.496,A -85,B 0,C 180,E1 -8848.182,E2 -8848.182} C_VEL
LIN {X 0,Y 446.41,Z 130.503,A -85,B 0,C 180,E1 -8851.301,E2 -8851.301} C_VEL
LIN {X 0,Y 446.422,Z 130.495,A -85,B 0,C 180,E1 -8854.524,E2 -8854.524} C_VEL
LIN {X 0,Y 446.405,Z 130.5,A -85,B 0,C 180,E1 -8858.077,E2 -8858.077} C_VEL
LIN {X 0,Y 446.401,Z 130.504,A -85,B 0,C 180,E1 -8861.394,E2 -8861.394} C_VEL
LIN {X 0,Y 446.45,Z 130.499,A -85,B 0,C 180,E1 -8865.104,E2 -8865.104} C_VEL
LIN {X 0,Y 446.401,Z 130.505,A -85,B 0,C 180,E1 -8868.606,E2 -8868.606} C_VEL
LIN {X 0,Y 446.398,Z 130.501,A -85,B 0,C 180,E1 -8871.924,E2 -8871.924} C_VEL
LIN {X 0,Y 446.414,Z 130.503,A -85,B 0,C 180,E1 -8875.476,E2 -8875.476} C_VEL
LIN {X 0,Y 446.388,Z 130.503,A -85,B 0,C 180,E1 -8878.697,E2 -8878.697} C_VEL
LIN {X 0,Y 446.422,Z 130.612,A -85,B 0,C 180,E1 -8881.929,E2 -8881.929} C_VEL
LIN {X 0,Y 449.664,Z 144.416,A -85,B 0,C 180,E1 -8884.696,E2 -8884.696} C_VEL
LIN {X 0,Y 453.707,Z 154.644,A -85,B 0,C 180,E1 -8885.115,E2 -8885.115} C_VEL
LIN {X 0,Y 456.551,Z 167.03,A -85,B 0,C 180,E1 -8885.492,E2 -8885.492} C_VEL
LIN {X 0,Y 455.713,Z 233.686,A -85,B 0,C 180,E1 -8886.572,E2 -8886.572} C_VEL
LIN {X 0,Y 454.88,Z 295.169,A -85,B 0,C 180,E1 -8887.56,E2 -8887.56} C_VEL
LIN {X 0,Y 454.195,Z 299.098,A -85,B 0,C 180,E1 -8887.59,E2 -8887.59} C_VEL
LIN {X 0,Y 448.547,Z 311.397,A -85,B 0,C 180,E1 -8887.539,E2 -8887.539} C_VEL
LIN {X 0,Y 447.88,Z 315.282,A -85,B 0,C 180,E1 -8887.608,E2 -8887.608} C_VEL
LIN {X 0,Y 447.321,Z 330.714,A -85,B 0,C 180,E1 -8888.117,E2 -8888.117} C_VEL
LIN {X 0,Y 446.553,Z 345.175,A -85,B 0,C 180,E1 -8888.778,E2 -8888.778} C_VEL
LIN {X 0,Y 445.693,Z 358.763,A -85,B 0,C 180,E1 -8889.581,E2 -8889.581} C_VEL
LIN {X 0,Y 444.6,Z 372.777,A -85,B 0,C 180,E1 -8890.612,E2 -8890.612} C_VEL
LIN {X 0,Y 443.616,Z 384.968,A -85,B 0,C 180,E1 -8891.714,E2 -8891.714} C_VEL
LIN {X 0,Y 442.604,Z 396.135,A -85,B 0,C 180,E1 -8892.917,E2 -8892.917} C_VEL
LIN {X 0,Y 441.655,Z 406.948,A -85,B 0,C 180,E1 -8894.305,E2 -8894.305} C_VEL
LIN {X 0,Y 440.673,Z 417.463,A -85,B 0,C 180,E1 -8895.924,E2 -8895.924} C_VEL
LIN {X 0,Y 439.994,Z 426.198,A -85,B 0,C 180,E1 -8897.547,E2 -8897.547} C_VEL
LIN {X 0,Y 439.45,Z 432.505,A -85,B 0,C 180,E1 -8898.936,E2 -8898.936} C_VEL
LIN {X 0,Y 438.975,Z 439.446,A -85,B 0,C 180,E1 -8900.787,E2 -8900.787} C_VEL
LIN {X 0,Y 438.674,Z 444.9,A -85,B 0,C 180,E1 -8902.636,E2 -8902.636} C_VEL
LIN {X 0,Y 438.501,Z 449.017,A -85,B 0,C 180,E1 -8904.482,E2 -8904.482} C_VEL
LIN {X 0,Y 438.344,Z 451.914,A -85,B 0,C 180,E1 -8906.323,E2 -8906.323} C_VEL
LIN {X 0,Y 438.298,Z 453.657,A -85,B 0,C 180,E1 -8908.162,E2 -8908.162} C_VEL
LIN {X 0,Y 438.253,Z 454.267,A -85,B 0,C 180,E1 -8910,E2 -8910} C_VEL
LIN {X 0,Y 438.298,Z 453.707,A -85,B 0,C 180,E1 -8911.838,E2 -8911.838} C_VEL
LIN {X 0,Y 438.344,Z 452.031,A -85,B 0,C 180,E1 -8913.677,E2 -8913.677} C_VEL
LIN {X 0,Y 438.495,Z 449.199,A -85,B 0,C 180,E1 -8915.518,E2 -8915.518} C_VEL
LIN {X 0,Y 438.664,Z 445.145,A -85,B 0,C 180,E1 -8917.364,E2 -8917.364} C_VEL
LIN {X 0,Y 438.964,Z 439.767,A -85,B 0,C 180,E1 -8919.213,E2 -8919.213} C_VEL
LIN {X 0,Y 439.437,Z 432.913,A -85,B 0,C 180,E1 -8921.065,E2 -8921.065} C_VEL
LIN {X 0,Y 440.008,Z 425.54,A -85,B 0,C 180,E1 -8922.687,E2 -8922.687} C_VEL
LIN {X 0,Y 440.757,Z 416.655,A -85,B 0,C 180,E1 -8924.309,E2 -8924.309} C_VEL
LIN {X 0,Y 441.579,Z 407.594,A -85,B 0,C 180,E1 -8925.698,E2 -8925.698} C_VEL
LIN {X 0,Y 442.552,Z 396.901,A -85,B 0,C 180,E1 -8927.085,E2 -8927.085} C_VEL
LIN {X 0,Y 443.569,Z 385.401,A -85,B 0,C 180,E1 -8928.337,E2 -8928.337} C_VEL
LIN {X 0,Y 444.538,Z 373.894,A -85,B 0,C 180,E1 -8929.391,E2 -8929.391} C_VEL
LIN {X 0,Y 445.566,Z 360.159,A -85,B 0,C 180,E1 -8930.425,E2 -8930.425} C_VEL
LIN {X 0,Y 446.61,Z 345.389,A -85,B 0,C 180,E1 -8931.303,E2 -8931.303} C_VEL
LIN {X 0,Y 447.323,Z 330.532,A -85,B 0,C 180,E1 -8931.985,E2 -8931.985} C_VEL
LIN {X 0,Y 447.874,Z 316.373,A -85,B 0,C 180,E1 -8932.458,E2 -8932.458} C_VEL
LIN {X 0,Y 448.285,Z 300.248,A -85,B 0,C 180,E1 -8932.801,E2 -8932.801} C_VEL
LIN {X 0,Y 450.193,Z 168.998,A -85,B 0,C 180,E1 -8934.943,E2 -8934.943} C_VEL
LIN {X 0,Y 447.079,Z 155.64,A -85,B 0,C 180,E1 -8935.363,E2 -8935.363} C_VEL
LIN {X 0,Y 442.434,Z 144.472,A -85,B 0,C 180,E1 -8935.865,E2 -8935.865} C_VEL
LIN {X 0,Y 439.374,Z 131.381,A -85,B 0,C 180,E1 -8938.558,E2 -8938.558} C_VEL
LIN {X 0,Y 439.346,Z 131.386,A -85,B 0,C 180,E1 -8941.863,E2 -8941.863} C_VEL
LIN {X 0,Y 439.383,Z 131.384,A -85,B 0,C 180,E1 -8945.338,E2 -8945.338} C_VEL
LIN {X 0,Y 439.348,Z 131.386,A -85,B 0,C 180,E1 -8948.599,E2 -8948.599} C_VEL
LIN {X 0,Y 439.345,Z 131.382,A -85,B 0,C 180,E1 -8952.211,E2 -8952.211} C_VEL
LIN {X 0,Y 439.373,Z 131.381,A -85,B 0,C 180,E1 -8955.267,E2 -8955.267} C_VEL
LIN {X 0,Y 439.355,Z 131.382,A -85,B 0,C 180,E1 -8959.016,E2 -8959.016} C_VEL
LIN {X 0,Y 439.357,Z 131.374,A -85,B 0,C 180,E1 -8961.611,E2 -8961.611} C_VEL
LIN {X 0,Y 439.393,Z 131.38,A -85,B 0,C 180,E1 -8964.843,E2 -8964.843} C_VEL
LIN {X 0,Y 439.355,Z 131.371,A -85,B 0,C 180,E1 -8968.138,E2 -8968.138} C_VEL
LIN {X 0,Y 439.386,Z 131.375,A -85,B 0,C 180,E1 -8971.61,E2 -8971.61} C_VEL
LIN {X 0,Y 439.368,Z 131.379,A -85,B 0,C 180,E1 -8974.413,E2 -8974.413} C_VEL
LIN {X 0,Y 439.362,Z 131.375,A -85,B 0,C 180,E1 -8977.424,E2 -8977.424} C_VEL
LIN {X 0,Y 439.443,Z 131.368,A -85,B 0,C 180,E1 -8980.663,E2 -8980.663} C_VEL
LIN {X 0,Y 439.422,Z 131.375,A -85,B 0,C 180,E1 -8984.223,E2 -8984.223} C_VEL
LIN {X 0,Y 439.488,Z 131.36,A -85,B 0,C 180,E1 -8987.285,E2 -8987.285} C_VEL
LIN {X 0,Y 439.493,Z 131.356,A -85,B 0,C 180,E1 -8990.798,E2 -8990.798} C_VEL
LIN {X 0,Y 439.562,Z 131.358,A -85,B 0,C 180,E1 -8993.574,E2 -8993.574} C_VEL
LIN {X 0,Y 439.41,Z 131.371,A -85,B 0,C 180,E1 -8995.413,E2 -8995.413} C_VEL
LIN {X 0,Y 439.629,Z 131.346,A -85,B 0,C 180,E1 -8998.168,E2 -8998.168} C_VEL
LIN {X 0,Y 439.713,Z 131.333,A -85,B 0,C 180,E1 -9000,E2 -9000} C_VEL
LIN {X 0,Y 439.633,Z 131.345,A -85,B 0,C 180,E1 -9002.749,E2 -9002.749} C_VEL
LIN {X 0,Y 439.567,Z 131.353,A -85,B 0,C 180,E1 -9006.426,E2 -9006.426} C_VEL
LIN {X 0,Y 439.497,Z 131.362,A -85,B 0,C 180,E1 -9009.202,E2 -9009.202} C_VEL
LIN {X 0,Y 439.468,Z 131.369,A -85,B 0,C 180,E1 -9012.937,E2 -9012.937} C_VEL
LIN {X 0,Y 439.449,Z 131.369,A -85,B 0,C 180,E1 -9016.348,E2 -9016.348} C_VEL
LIN {X 0,Y 439.404,Z 131.376,A -85,B 0,C 180,E1 -9019.626,E2 -9019.626} C_VEL
LIN {X 0,Y 439.365,Z 131.377,A -85,B 0,C 180,E1 -9022.575,E2 -9022.575} C_VEL
LIN {X 0,Y 439.379,Z 131.375,A -85,B 0,C 180,E1 -9025.586,E2 -9025.586} C_VEL
LIN {X 0,Y 439.402,Z 131.38,A -85,B 0,C 180,E1 -9028.674,E2 -9028.674} C_VEL
LIN {X 0,Y 439.37,Z 131.378,A -85,B 0,C 180,E1 -9032.03,E2 -9032.03} C_VEL
LIN {X 0,Y 439.394,Z 131.375,A -85,B 0,C 180,E1 -9035.34,E2 -9035.34} C_VEL
LIN {X 0,Y 439.377,Z 131.382,A -85,B 0,C 180,E1 -9038.596,E2 -9038.596} C_VEL
LIN {X 0,Y 439.39,Z 131.376,A -85,B 0,C 180,E1 -9041.256,E2 -9041.256} C_VEL
LIN {X 0,Y 439.401,Z 131.375,A -85,B 0,C 180,E1 -9044.729,E2 -9044.729} C_VEL
LIN {X 0,Y 439.397,Z 131.375,A -85,B 0,C 180,E1 -9047.795,E2 -9047.795} C_VEL
LIN {X 0,Y 439.431,Z 131.365,A -85,B 0,C 180,E1 -9050.228,E2 -9050.228} C_VEL
LIN {X 0,Y 439.374,Z 131.379,A -85,B 0,C 180,E1 -9053.713,E2 -9053.713} C_VEL
LIN {X 0,Y 439.373,Z 131.38,A -85,B 0,C 180,E1 -9057.054,E2 -9057.054} C_VEL
LIN {X 0,Y 439.396,Z 131.536,A -85,B 0,C 180,E1 -9058.209,E2 -9058.209} C_VEL
LIN {X 0,Y 443.204,Z 146.453,A -85,B 0,C 180,E1 -9060.994,E2 -9060.994} C_VEL
LIN {X 0,Y 444.915,Z 154.565,A -85,B 0,C 180,E1 -9062.438,E2 -9062.438} C_VEL
LIN {X 0,Y 444.108,Z 166.26,A -85,B 0,C 180,E1 -9064.287,E2 -9064.287} C_VEL
LIN {X 0,Y 449.9,Z 195.86,A -85,B 0,C 180,E1 -9065.154,E2 -9065.154} C_VEL
LIN {X 0,Y 447.87,Z 331.979,A -85,B 0,C 180,E1 -9067.39,E2 -9067.39} C_VEL
LIN {X 0,Y 447.265,Z 347.533,A -85,B 0,C 180,E1 -9067.814,E2 -9067.814} C_VEL
LIN {X 0,Y 446.468,Z 362.077,A -85,B 0,C 180,E1 -9068.391,E2 -9068.391} C_VEL
LIN {X 0,Y 445.627,Z 375.523,A -85,B 0,C 180,E1 -9069.095,E2 -9069.095} C_VEL
LIN {X 0,Y 444.543,Z 389.432,A -85,B 0,C 180,E1 -9070.008,E2 -9070.008} C_VEL
LIN {X 0,Y 443.523,Z 402.179,A -85,B 0,C 180,E1 -9071.044,E2 -9071.044} C_VEL
LIN {X 0,Y 442.56,Z 414.001,A -85,B 0,C 180,E1 -9072.2,E2 -9072.2} C_VEL
LIN {X 0,Y 441.519,Z 425.874,A -85,B 0,C 180,E1 -9073.588,E2 -9073.588} C_VEL
LIN {X 0,Y 440.599,Z 435.867,A -85,B 0,C 180,E1 -9074.977,E2 -9074.977} C_VEL
LIN {X 0,Y 439.759,Z 445.646,A -85,B 0,C 180,E1 -9076.601,E2 -9076.601} C_VEL
LIN {X 0,Y 439.231,Z 453.812,A -85,B 0,C 180,E1 -9078.228,E2 -9078.228} C_VEL
LIN {X 0,Y 438.774,Z 460.561,A -85,B 0,C 180,E1 -9079.852,E2 -9079.852} C_VEL
LIN {X 0,Y 438.54,Z 466.8,A -85,B 0,C 180,E1 -9081.707,E2 -9081.707} C_VEL
LIN {X 0,Y 438.363,Z 472.013,A -85,B 0,C 180,E1 -9083.723,E2 -9083.723} C_VEL
LIN {X 0,Y 438.284,Z 475.16,A -85,B 0,C 180,E1 -9085.401,E2 -9085.401} C_VEL
LIN {X 0,Y 438.324,Z 477.488,A -85,B 0,C 180,E1 -9087.243,E2 -9087.243} C_VEL
LIN {X 0,Y 438.249,Z 478.657,A -85,B 0,C 180,E1 -9089.081,E2 -9089.081} C_VEL
LIN {X 0,Y 438.249,Z 478.655,A -85,B 0,C 180,E1 -9090.919,E2 -9090.919} C_VEL
LIN {X 0,Y 438.324,Z 477.482,A -85,B 0,C 180,E1 -9092.757,E2 -9092.757} C_VEL
LIN {X 0,Y 438.285,Z 475.151,A -85,B 0,C 180,E1 -9094.599,E2 -9094.599} C_VEL
LIN {X 0,Y 438.396,Z 471.62,A -85,B 0,C 180,E1 -9096.443,E2 -9096.443} C_VEL
LIN {X 0,Y 438.539,Z 466.794,A -85,B 0,C 180,E1 -9098.293,E2 -9098.293} C_VEL
LIN {X 0,Y 438.774,Z 460.545,A -85,B 0,C 180,E1 -9100.148,E2 -9100.148} C_VEL
LIN {X 0,Y 439.214,Z 453.791,A -85,B 0,C 180,E1 -9101.772,E2 -9101.772} C_VEL
LIN {X 0,Y 439.759,Z 445.626,A -85,B 0,C 180,E1 -9103.399,E2 -9103.399} C_VEL
LIN {X 0,Y 440.599,Z 435.844,A -85,B 0,C 180,E1 -9105.023,E2 -9105.023} C_VEL
LIN {X 0,Y 441.469,Z 425.843,A -85,B 0,C 180,E1 -9106.414,E2 -9106.414} C_VEL
LIN {X 0,Y 442.511,Z 413.97,A -85,B 0,C 180,E1 -9107.802,E2 -9107.802} C_VEL
LIN {X 0,Y 443.479,Z 402.139,A -85,B 0,C 180,E1 -9108.958,E2 -9108.958} C_VEL
LIN {X 0,Y 444.546,Z 389.368,A -85,B 0,C 180,E1 -9109.991,E2 -9109.991} C_VEL
LIN {X 0,Y 445.614,Z 375.439,A -85,B 0,C 180,E1 -9110.906,E2 -9110.906} C_VEL
LIN {X 0,Y 446.561,Z 361.244,A -85,B 0,C 180,E1 -9111.639,E2 -9111.639} C_VEL
LIN {X 0,Y 447.25,Z 347.403,A -85,B 0,C 180,E1 -9112.187,E2 -9112.187} C_VEL
LIN {X 0,Y 447.839,Z 331.734,A -85,B 0,C 180,E1 -9112.612,E2 -9112.612} C_VEL
LIN {X 0,Y 449.835,Z 200.136,A -85,B 0,C 180,E1 -9114.771,E2 -9114.771} C_VEL
LIN {X 0,Y 449.759,Z 194.839,A -85,B 0,C 180,E1 -9114.867,E2 -9114.867} C_VEL
LIN {X 0,Y 444.152,Z 166.24,A -85,B 0,C 180,E1 -9115.706,E2 -9115.706} C_VEL
LIN {X 0,Y 444.912,Z 154.566,A -85,B 0,C 180,E1 -9117.555,E2 -9117.555} C_VEL
LIN {X 0,Y 442.158,Z 142.164,A -85,B 0,C 180,E1 -9119.783,E2 -9119.783} C_VEL
LIN {X 0,Y 439.373,Z 131.379,A -85,B 0,C 180,E1 -9121.827,E2 -9121.827} C_VEL
LIN {X 0,Y 439.4,Z 131.373,A -85,B 0,C 180,E1 -9125.156,E2 -9125.156} C_VEL
LIN {X 0,Y 439.386,Z 131.377,A -85,B 0,C 180,E1 -9128.595,E2 -9128.595} C_VEL
LIN {X 0,Y 439.389,Z 131.376,A -85,B 0,C 180,E1 -9131.257,E2 -9131.257} C_VEL
LIN {X 0,Y 439.401,Z 131.372,A -85,B 0,C 180,E1 -9134.73,E2 -9134.73} C_VEL
LIN {X 0,Y 439.397,Z 131.378,A -85,B 0,C 180,E1 -9137.796,E2 -9137.796} C_VEL
LIN {X 0,Y 439.396,Z 131.374,A -85,B 0,C 180,E1 -9140.224,E2 -9140.224} C_VEL
LIN {X 0,Y 439.374,Z 131.376,A -85,B 0,C 180,E1 -9143.713,E2 -9143.713} C_VEL
LIN {X 0,Y 439.373,Z 131.377,A -85,B 0,C 180,E1 -9147.054,E2 -9147.054} C_VEL
LIN {X 0,Y 439.382,Z 131.372,A -85,B 0,C 180,E1 -9150.274,E2 -9150.274} C_VEL
LIN {X 0,Y 439.42,Z 131.373,A -85,B 0,C 180,E1 -9153.396,E2 -9153.396} C_VEL
LIN {X 0,Y 439.383,Z 131.374,A -85,B 0,C 180,E1 -9156.43,E2 -9156.43} C_VEL
LIN {X 0,Y 439.39,Z 131.373,A -85,B 0,C 180,E1 -9159.397,E2 -9159.397} C_VEL
LIN {X 0,Y 439.406,Z 131.374,A -85,B 0,C 180,E1 -9162.309,E2 -9162.309} C_VEL
LIN {X 0,Y 439.448,Z 131.371,A -85,B 0,C 180,E1 -9165.174,E2 -9165.174} C_VEL
LIN {X 0,Y 439.486,Z 131.359,A -85,B 0,C 180,E1 -9168.001,E2 -9168.001} C_VEL
LIN {X 0,Y 439.506,Z 131.355,A -85,B 0,C 180,E1 -9171.726,E2 -9171.726} C_VEL
LIN {X 0,Y 439.607,Z 131.353,A -85,B 0,C 180,E1 -9174.496,E2 -9174.496} C_VEL
LIN {X 0,Y 439.635,Z 131.348,A -85,B 0,C 180,E1 -9178.168,E2 -9178.168} C_VEL
LIN {X 0,Y 439.712,Z 131.335,A -85,B 0,C 180,E1 -9180,E2 -9180} C_VEL
LIN {X 0,Y 439.609,Z 131.349,A -85,B 0,C 180,E1 -9182.749,E2 -9182.749} C_VEL
LIN {X 0,Y 439.565,Z 131.358,A -85,B 0,C 180,E1 -9186.426,E2 -9186.426} C_VEL
LIN {X 0,Y 439.493,Z 131.357,A -85,B 0,C 180,E1 -9189.202,E2 -9189.202} C_VEL
LIN {X 0,Y 439.467,Z 131.36,A -85,B 0,C 180,E1 -9192.938,E2 -9192.938} C_VEL
LIN {X 0,Y 439.404,Z 131.372,A -85,B 0,C 180,E1 -9196.328,E2 -9196.328} C_VEL
LIN {X 0,Y 439.404,Z 131.378,A -85,B 0,C 180,E1 -9199.626,E2 -9199.626} C_VEL
LIN {X 0,Y 439.365,Z 131.378,A -85,B 0,C 180,E1 -9202.576,E2 -9202.576} C_VEL
LIN {X 0,Y 439.368,Z 131.368,A -85,B 0,C 180,E1 -9205.587,E2 -9205.587} C_VEL
LIN {X 0,Y 439.391,Z 131.373,A -85,B 0,C 180,E1 -9208.675,E2 -9208.675} C_VEL
LIN {X 0,Y 439.367,Z 131.379,A -85,B 0,C 180,E1 -9212.029,E2 -9212.029} C_VEL
LIN {X 0,Y 439.391,Z 131.378,A -85,B 0,C 180,E1 -9215.339,E2 -9215.339} C_VEL
LIN {X 0,Y 439.358,Z 131.378,A -85,B 0,C 180,E1 -9218.598,E2 -9218.598} C_VEL
LIN {X 0,Y 439.349,Z 131.376,A -85,B 0,C 180,E1 -9222.21,E2 -9222.21} C_VEL
LIN {X 0,Y 439.398,Z 131.379,A -85,B 0,C 180,E1 -9225.27,E2 -9225.27} C_VEL
LIN {X 0,Y 439.354,Z 131.384,A -85,B 0,C 180,E1 -9229.016,E2 -9229.016} C_VEL
LIN {X 0,Y 439.356,Z 131.378,A -85,B 0,C 180,E1 -9231.611,E2 -9231.611} C_VEL
LIN {X 0,Y 439.389,Z 131.376,A -85,B 0,C 180,E1 -9234.843,E2 -9234.843} C_VEL
LIN {X 0,Y 439.346,Z 131.384,A -85,B 0,C 180,E1 -9238.137,E2 -9238.137} C_VEL
LIN {X 0,Y 439.353,Z 131.378,A -85,B 0,C 180,E1 -9241.322,E2 -9241.322} C_VEL
LIN {X 0,Y 439.374,Z 131.421,A -85,B 0,C 180,E1 -9241.555,E2 -9241.555} C_VEL
LIN {X 0,Y 442.482,Z 144.592,A -85,B 0,C 180,E1 -9244.254,E2 -9244.254} C_VEL
LIN {X 0,Y 447.656,Z 157.535,A -85,B 0,C 180,E1 -9244.801,E2 -9244.801} C_VEL
LIN {X 0,Y 450.112,Z 168.34,A -85,B 0,C 180,E1 -9245.137,E2 -9245.137} C_VEL
LIN {X 0,Y 449.223,Z 233.911,A -85,B 0,C 180,E1 -9246.213,E2 -9246.213} C_VEL
LIN {X 0,Y 448.061,Z 309.336,A -85,B 0,C 180,E1 -9247.461,E2 -9247.461} C_VEL
LIN {X 0,Y 447.88,Z 315.282,A -85,B 0,C 180,E1 -9247.608,E2 -9247.608} C_VEL
LIN {X 0,Y 447.221,Z 321.04,A -85,B 0,C 180,E1 -9247.745,E2 -9247.745} C_VEL
LIN {X 0,Y 444.294,Z 330.368,A -85,B 0,C 180,E1 -9247.939,E2 -9247.939} C_VEL
LIN {X 0,Y 441.069,Z 339.58,A -85,B 0,C 180,E1 -9248.19,E2 -9248.19} C_VEL
LIN {X 0,Y 439.976,Z 345.074,A -85,B 0,C 180,E1 -9248.428,E2 -9248.428} C_VEL
LIN {X 0,Y 439.029,Z 358.969,A -85,B 0,C 180,E1 -9249.257,E2 -9249.257} C_VEL
LIN {X 0,Y 437.906,Z 372.981,A -85,B 0,C 180,E1 -9250.304,E2 -9250.304} C_VEL
LIN {X 0,Y 436.82,Z 385.525,A -85,B 0,C 180,E1 -9251.456,E2 -9251.456} C_VEL
LIN {X 0,Y 435.783,Z 396.338,A -85,B 0,C 180,E1 -9252.641,E2 -9252.641} C_VEL
LIN {X 0,Y 434.803,Z 407.151,A -85,B 0,C 180,E1 -9254.051,E2 -9254.051} C_VEL
LIN {X 0,Y 433.768,Z 417.665,A -85,B 0,C 180,E1 -9255.695,E2 -9255.695} C_VEL
LIN {X 0,Y 433.019,Z 426.478,A -85,B 0,C 180,E1 -9257.36,E2 -9257.36} C_VEL
LIN {X 0,Y 432.471,Z 432.706,A -85,B 0,C 180,E1 -9258.755,E2 -9258.755} C_VEL
LIN {X 0,Y 431.945,Z 439.647,A -85,B 0,C 180,E1 -9260.636,E2 -9260.636} C_VEL
LIN {X 0,Y 431.616,Z 445.1,A -85,B 0,C 180,E1 -9262.515,E2 -9262.515} C_VEL
LIN {X 0,Y 431.425,Z 449.217,A -85,B 0,C 180,E1 -9264.391,E2 -9264.391} C_VEL
LIN {X 0,Y 431.249,Z 452.113,A -85,B 0,C 180,E1 -9266.262,E2 -9266.262} C_VEL
LIN {X 0,Y 431.222,Z 453.855,A -85,B 0,C 180,E1 -9268.132,E2 -9268.132} C_VEL
LIN {X 0,Y 431.167,Z 454.466,A -85,B 0,C 180,E1 -9270,E2 -9270} C_VEL
LIN {X 0,Y 431.222,Z 453.905,A -85,B 0,C 180,E1 -9271.868,E2 -9271.868} C_VEL
LIN {X 0,Y 431.248,Z 452.23,A -85,B 0,C 180,E1 -9273.738,E2 -9273.738} C_VEL
LIN {X 0,Y 431.42,Z 449.397,A -85,B 0,C 180,E1 -9275.609,E2 -9275.609} C_VEL
LIN {X 0,Y 431.607,Z 445.343,A -85,B 0,C 180,E1 -9277.485,E2 -9277.485} C_VEL
LIN {X 0,Y 431.934,Z 439.965,A -85,B 0,C 180,E1 -9279.364,E2 -9279.364} C_VEL
LIN {X 0,Y 432.458,Z 433.11,A -85,B 0,C 180,E1 -9281.246,E2 -9281.246} C_VEL
LIN {X 0,Y 433.029,Z 425.78,A -85,B 0,C 180,E1 -9282.886,E2 -9282.886} C_VEL
LIN {X 0,Y 433.856,Z 416.852,A -85,B 0,C 180,E1 -9284.542,E2 -9284.542} C_VEL
LIN {X 0,Y 434.736,Z 407.79,A -85,B 0,C 180,E1 -9285.952,E2 -9285.952} C_VEL
LIN {X 0,Y 435.762,Z 397.097,A -85,B 0,C 180,E1 -9287.36,E2 -9287.36} C_VEL
LIN {X 0,Y 436.829,Z 385.38,A -85,B 0,C 180,E1 -9288.653,E2 -9288.653} C_VEL
LIN {X 0,Y 437.959,Z 372.668,A -85,B 0,C 180,E1 -9289.816,E2 -9289.816} C_VEL
LIN {X 0,Y 439.082,Z 358.59,A -85,B 0,C 180,E1 -9290.863,E2 -9290.863} C_VEL
LIN {X 0,Y 440.082,Z 344.185,A -85,B 0,C 180,E1 -9291.711,E2 -9291.711} C_VEL
LIN {X 0,Y 440.823,Z 329.432,A -85,B 0,C 180,E1 -9292.378,E2 -9292.378} C_VEL
LIN {X 0,Y 441.418,Z 314.278,A -85,B 0,C 180,E1 -9292.866,E2 -9292.866} C_VEL
LIN {X 0,Y 441.836,Z 295.059,A -85,B 0,C 180,E1 -9293.246,E2 -9293.246} C_VEL
LIN {X 0,Y 443.766,Z 169.965,A -85,B 0,C 180,E1 -9295.316,E2 -9295.316} C_VEL
LIN {X 0,Y 441.016,Z 158.419,A -85,B 0,C 180,E1 -9295.691,E2 -9295.691} C_VEL
LIN {X 0,Y 435.291,Z 144.703,A -85,B 0,C 180,E1 -9296.318,E2 -9296.318} C_VEL
LIN {X 0,Y 432.316,Z 132.26,A -85,B 0,C 180,E1 -9298.942,E2 -9298.942} C_VEL
LIN {X 0,Y 432.3,Z 132.264,A -85,B 0,C 180,E1 -9301.348,E2 -9301.348} C_VEL
LIN {X 0,Y 432.322,Z 132.259,A -85,B 0,C 180,E1 -9304.679,E2 -9304.679} C_VEL
LIN {X 0,Y 432.318,Z 132.26,A -85,B 0,C 180,E1 -9308.152,E2 -9308.152} C_VEL
LIN {X 0,Y 432.301,Z 132.26,A -85,B 0,C 180,E1 -9311.801,E2 -9311.801} C_VEL
LIN {X 0,Y 432.333,Z 132.256,A -85,B 0,C 180,E1 -9314.348,E2 -9314.348} C_VEL
LIN {X 0,Y 432.301,Z 132.252,A -85,B 0,C 180,E1 -9317.019,E2 -9317.019} C_VEL
LIN {X 0,Y 432.289,Z 132.26,A -85,B 0,C 180,E1 -9319.828,E2 -9319.828} C_VEL
LIN {X 0,Y 432.297,Z 132.251,A -85,B 0,C 180,E1 -9323.021,E2 -9323.021} C_VEL
LIN {X 0,Y 432.334,Z 132.255,A -85,B 0,C 180,E1 -9326.002,E2 -9326.002} C_VEL
LIN {X 0,Y 432.333,Z 132.243,A -85,B 0,C 180,E1 -9329.494,E2 -9329.494} C_VEL
LIN {X 0,Y 432.316,Z 132.257,A -85,B 0,C 180,E1 -9331.872,E2 -9331.872} C_VEL
LIN {X 0,Y 432.326,Z 132.256,A -85,B 0,C 180,E1 -9334.997,E2 -9334.997} C_VEL
LIN {X 0,Y 432.357,Z 132.25,A -85,B 0,C 180,E1 -9338.046,E2 -9338.046} C_VEL
LIN {X 0,Y 432.383,Z 132.245,A -85,B 0,C 180,E1 -9341.029,E2 -9341.029} C_VEL
LIN {X 0,Y 432.391,Z 132.251,A -85,B 0,C 180,E1 -9343.96,E2 -9343.96} C_VEL
LIN {X 0,Y 432.462,Z 132.24,A -85,B 0,C 180,E1 -9347.803,E2 -9347.803} C_VEL
LIN {X 0,Y 432.465,Z 132.235,A -85,B 0,C 180,E1 -9351.59,E2 -9351.59} C_VEL
LIN {X 0,Y 432.556,Z 132.223,A -85,B 0,C 180,E1 -9354.405,E2 -9354.405} C_VEL
LIN {X 0,Y 432.599,Z 132.222,A -85,B 0,C 180,E1 -9358.138,E2 -9358.138} C_VEL
LIN {X 0,Y 432.663,Z 132.211,A -85,B 0,C 180,E1 -9360,E2 -9360} C_VEL
LIN {X 0,Y 432.584,Z 132.223,A -85,B 0,C 180,E1 -9362.794,E2 -9362.794} C_VEL
LIN {X 0,Y 432.58,Z 132.225,A -85,B 0,C 180,E1 -9365.594,E2 -9365.594} C_VEL
LIN {X 0,Y 432.466,Z 132.235,A -85,B 0,C 180,E1 -9368.41,E2 -9368.41} C_VEL
LIN {X 0,Y 432.462,Z 132.238,A -85,B 0,C 180,E1 -9372.196,E2 -9372.196} C_VEL
LIN {X 0,Y 432.432,Z 132.243,A -85,B 0,C 180,E1 -9376.039,E2 -9376.039} C_VEL
LIN {X 0,Y 432.389,Z 132.251,A -85,B 0,C 180,E1 -9379.485,E2 -9379.485} C_VEL
LIN {X 0,Y 432.319,Z 132.257,A -85,B 0,C 180,E1 -9382.964,E2 -9382.964} C_VEL
LIN {X 0,Y 432.339,Z 132.257,A -85,B 0,C 180,E1 -9385.002,E2 -9385.002} C_VEL
LIN {X 0,Y 432.349,Z 132.253,A -85,B 0,C 180,E1 -9388.125,E2 -9388.125} C_VEL
LIN {X 0,Y 432.322,Z 132.257,A -85,B 0,C 180,E1 -9391.346,E2 -9391.346} C_VEL
LIN {X 0,Y 432.339,Z 132.256,A -85,B 0,C 180,E1 -9394.677,E2 -9394.677} C_VEL
LIN {X 0,Y 432.336,Z 132.255,A -85,B 0,C 180,E1 -9398.15,E2 -9398.15} C_VEL
LIN {X 0,Y 432.334,Z 132.255,A -85,B 0,C 180,E1 -9401.602,E2 -9401.602} C_VEL
LIN {X 0,Y 432.335,Z 132.258,A -85,B 0,C 180,E1 -9404.347,E2 -9404.347} C_VEL
LIN {X 0,Y 432.321,Z 132.255,A -85,B 0,C 180,E1 -9407.015,E2 -9407.015} C_VEL
LIN {X 0,Y 432.337,Z 132.247,A -85,B 0,C 180,E1 -9409.82,E2 -9409.82} C_VEL
LIN {X 0,Y 432.307,Z 132.258,A -85,B 0,C 180,E1 -9413.022,E2 -9413.022} C_VEL
LIN {X 0,Y 432.36,Z 132.256,A -85,B 0,C 180,E1 -9415.996,E2 -9415.996} C_VEL
LIN {X 0,Y 432.323,Z 132.28,A -85,B 0,C 180,E1 -9417.791,E2 -9417.791} C_VEL
LIN {X 0,Y 436.265,Z 147.721,A -85,B 0,C 180,E1 -9420.736,E2 -9420.736} C_VEL
LIN {X 0,Y 438.089,Z 156.195,A -85,B 0,C 180,E1 -9422.275,E2 -9422.275} C_VEL
LIN {X 0,Y 437.475,Z 166.288,A -85,B 0,C 180,E1 -9423.876,E2 -9423.876} C_VEL
LIN {X 0,Y 443.463,Z 196.841,A -85,B 0,C 180,E1 -9424.788,E2 -9424.788} C_VEL
LIN {X 0,Y 441.315,Z 331.796,A -85,B 0,C 180,E1 -9427.035,E2 -9427.035} C_VEL
LIN {X 0,Y 440.697,Z 347.344,A -85,B 0,C 180,E1 -9427.465,E2 -9427.465} C_VEL
LIN {X 0,Y 439.872,Z 361.816,A -85,B 0,C 180,E1 -9428.047,E2 -9428.047} C_VEL
LIN {X 0,Y 438.989,Z 375.329,A -85,B 0,C 180,E1 -9428.764,E2 -9428.764} C_VEL
LIN {X 0,Y 437.824,Z 389.236,A -85,B 0,C 180,E1 -9429.688,E2 -9429.688} C_VEL
LIN {X 0,Y 436.757,Z 401.982,A -85,B 0,C 180,E1 -9430.739,E2 -9430.739} C_VEL
LIN {X 0,Y 435.74,Z 413.803,A -85,B 0,C 180,E1 -9431.912,E2 -9431.912} C_VEL
LIN {X 0,Y 434.647,Z 425.676,A -85,B 0,C 180,E1 -9433.321,E2 -9433.321} C_VEL
LIN {X 0,Y 433.648,Z 435.667,A -85,B 0,C 180,E1 -9434.73,E2 -9434.73} C_VEL
LIN {X 0,Y 432.794,Z 445.447,A -85,B 0,C 180,E1 -9436.381,E2 -9436.381} C_VEL
LIN {X 0,Y 432.214,Z 453.612,A -85,B 0,C 180,E1 -9438.034,E2 -9438.034} C_VEL
LIN {X 0,Y 431.732,Z 460.362,A -85,B 0,C 180,E1 -9439.685,E2 -9439.685} C_VEL
LIN {X 0,Y 431.45,Z 466.6,A -85,B 0,C 180,E1 -9441.57,E2 -9441.57} C_VEL
LIN {X 0,Y 431.287,Z 471.426,A -85,B 0,C 180,E1 -9443.45,E2 -9443.45} C_VEL
LIN {X 0,Y 431.208,Z 474.962,A -85,B 0,C 180,E1 -9445.326,E2 -9445.326} C_VEL
LIN {X 0,Y 431.217,Z 477.289,A -85,B 0,C 180,E1 -9447.197,E2 -9447.197} C_VEL
LIN {X 0,Y 431.165,Z 478.458,A -85,B 0,C 180,E1 -9449.066,E2 -9449.066} C_VEL
LIN {X 0,Y 431.165,Z 478.457,A -85,B 0,C 180,E1 -9450.934,E2 -9450.934} C_VEL
LIN {X 0,Y 431.217,Z 477.282,A -85,B 0,C 180,E1 -9452.803,E2 -9452.803} C_VEL
LIN {X 0,Y 431.21,Z 474.952,A -85,B 0,C 180,E1 -9454.674,E2 -9454.674} C_VEL
LIN {X 0,Y 431.324,Z 471.42,A -85,B 0,C 180,E1 -9456.549,E2 -9456.549} C_VEL
LIN {X 0,Y 431.45,Z 466.593,A -85,B 0,C 180,E1 -9458.43,E2 -9458.43} C_VEL
LIN {X 0,Y 431.731,Z 460.344,A -85,B 0,C 180,E1 -9460.315,E2 -9460.315} C_VEL
LIN {X 0,Y 432.205,Z 453.589,A -85,B 0,C 180,E1 -9461.966,E2 -9461.966} C_VEL
LIN {X 0,Y 432.902,Z 444.16,A -85,B 0,C 180,E1 -9463.855,E2 -9463.855} C_VEL
LIN {X 0,Y 433.776,Z 434.117,A -85,B 0,C 180,E1 -9465.506,E2 -9465.506} C_VEL
LIN {X 0,Y 434.761,Z 423.849,A -85,B 0,C 180,E1 -9466.916,E2 -9466.916} C_VEL
LIN {X 0,Y 435.849,Z 411.616,A -85,B 0,C 180,E1 -9468.327,E2 -9468.327} C_VEL
LIN {X 0,Y 436.983,Z 399.343,A -85,B 0,C 180,E1 -9469.495,E2 -9469.495} C_VEL
LIN {X 0,Y 438.121,Z 385.989,A -85,B 0,C 180,E1 -9470.543,E2 -9470.543} C_VEL
LIN {X 0,Y 439.237,Z 371.253,A -85,B 0,C 180,E1 -9471.47,E2 -9471.47} C_VEL
LIN {X 0,Y 440.226,Z 355.698,A -85,B 0,C 180,E1 -9472.219,E2 -9472.219} C_VEL
LIN {X 0,Y 440.991,Z 339.754,A -85,B 0,C 180,E1 -9472.766,E2 -9472.766} C_VEL
LIN {X 0,Y 441.476,Z 323.801,A -85,B 0,C 180,E1 -9473.111,E2 -9473.111} C_VEL
LIN {X 0,Y 443.403,Z 196.333,A -85,B 0,C 180,E1 -9475.218,E2 -9475.218} C_VEL
LIN {X 0,Y 437.435,Z 166.179,A -85,B 0,C 180,E1 -9476.121,E2 -9476.121} C_VEL
LIN {X 0,Y 438.077,Z 156.149,A -85,B 0,C 180,E1 -9477.726,E2 -9477.726} C_VEL
LIN {X 0,Y 435.224,Z 143.528,A -85,B 0,C 180,E1 -9480.039,E2 -9480.039} C_VEL
LIN {X 0,Y 432.323,Z 132.251,A -85,B 0,C 180,E1 -9482.209,E2 -9482.209} C_VEL
LIN {X 0,Y 432.34,Z 132.252,A -85,B 0,C 180,E1 -9484.677,E2 -9484.677} C_VEL
LIN {X 0,Y 432.34,Z 132.258,A -85,B 0,C 180,E1 -9488.15,E2 -9488.15} C_VEL
LIN {X 0,Y 432.334,Z 132.258,A -85,B 0,C 180,E1 -9491.602,E2 -9491.602} C_VEL
LIN {X 0,Y 432.334,Z 132.253,A -85,B 0,C 180,E1 -9494.347,E2 -9494.347} C_VEL
LIN {X 0,Y 432.321,Z 132.255,A -85,B 0,C 180,E1 -9497.016,E2 -9497.016} C_VEL
LIN {X 0,Y 432.334,Z 132.257,A -85,B 0,C 180,E1 -9499.821,E2 -9499.821} C_VEL
LIN {X 0,Y 432.307,Z 132.258,A -85,B 0,C 180,E1 -9503.022,E2 -9503.022} C_VEL
LIN {X 0,Y 432.359,Z 132.249,A -85,B 0,C 180,E1 -9505.997,E2 -9505.997} C_VEL
LIN {X 0,Y 432.348,Z 132.251,A -85,B 0,C 180,E1 -9509.49,E2 -9509.49} C_VEL
LIN {X 0,Y 432.387,Z 132.249,A -85,B 0,C 180,E1 -9512.928,E2 -9512.928} C_VEL
LIN {X 0,Y 432.367,Z 132.247,A -85,B 0,C 180,E1 -9516.023,E2 -9516.023} C_VEL
LIN {X 0,Y 432.352,Z 132.254,A -85,B 0,C 180,E1 -9519.046,E2 -9519.046} C_VEL
LIN {X 0,Y 432.362,Z 132.25,A -85,B 0,C 180,E1 -9522.011,E2 -9522.011} C_VEL
LIN {X 0,Y 432.396,Z 132.251,A -85,B 0,C 180,E1 -9524.927,E2 -9524.927} C_VEL
LIN {X 0,Y 432.461,Z 132.233,A -85,B 0,C 180,E1 -9527.804,E2 -9527.804} C_VEL
LIN {X 0,Y 432.466,Z 132.232,A -85,B 0,C 180,E1 -9531.59,E2 -9531.59} C_VEL
LIN {X 0,Y 432.58,Z 132.229,A -85,B 0,C 180,E1 -9534.406,E2 -9534.406} C_VEL
LIN {X 0,Y 432.604,Z 132.223,A -85,B 0,C 180,E1 -9538.138,E2 -9538.138} C_VEL
LIN {X 0,Y 432.663,Z 132.213,A -85,B 0,C 180,E1 -9540,E2 -9540} C_VEL
LIN {X 0,Y 432.563,Z 132.226,A -85,B 0,C 180,E1 -9542.794,E2 -9542.794} C_VEL
LIN {X 0,Y 432.579,Z 132.221,A -85,B 0,C 180,E1 -9545.594,E2 -9545.594} C_VEL
LIN {X 0,Y 432.464,Z 132.236,A -85,B 0,C 180,E1 -9548.41,E2 -9548.41} C_VEL
LIN {X 0,Y 432.462,Z 132.238,A -85,B 0,C 180,E1 -9552.197,E2 -9552.197} C_VEL
LIN {X 0,Y 432.391,Z 132.249,A -85,B 0,C 180,E1 -9556.04,E2 -9556.04} C_VEL
LIN {X 0,Y 432.389,Z 132.25,A -85,B 0,C 180,E1 -9559.485,E2 -9559.485} C_VEL
LIN {X 0,Y 432.314,Z 132.257,A -85,B 0,C 180,E1 -9562.965,E2 -9562.965} C_VEL
LIN {X 0,Y 432.319,Z 132.241,A -85,B 0,C 180,E1 -9566.036,E2 -9566.036} C_VEL
LIN {X 0,Y 432.327,Z 132.255,A -85,B 0,C 180,E1 -9569.189,E2 -9569.189} C_VEL
LIN {X 0,Y 432.323,Z 132.255,A -85,B 0,C 180,E1 -9572.443,E2 -9572.443} C_VEL
LIN {X 0,Y 432.337,Z 132.255,A -85,B 0,C 180,E1 -9575.818,E2 -9575.818} C_VEL
LIN {X 0,Y 432.302,Z 132.259,A -85,B 0,C 180,E1 -9579.348,E2 -9579.348} C_VEL
LIN {X 0,Y 432.304,Z 132.255,A -85,B 0,C 180,E1 -9581.801,E2 -9581.801} C_VEL
LIN {X 0,Y 432.334,Z 132.253,A -85,B 0,C 180,E1 -9584.347,E2 -9584.347} C_VEL
LIN {X 0,Y 432.303,Z 132.261,A -85,B 0,C 180,E1 -9587.018,E2 -9587.018} C_VEL
LIN {X 0,Y 432.289,Z 132.262,A -85,B 0,C 180,E1 -9589.828,E2 -9589.828} C_VEL
LIN {X 0,Y 432.297,Z 132.265,A -85,B 0,C 180,E1 -9593.021,E2 -9593.021} C_VEL
LIN {X 0,Y 432.331,Z 132.257,A -85,B 0,C 180,E1 -9596.002,E2 -9596.002} C_VEL
LIN {X 0,Y 432.331,Z 132.243,A -85,B 0,C 180,E1 -9599.494,E2 -9599.494} C_VEL
LIN {X 0,Y 432.336,Z 132.33,A -85,B 0,C 180,E1 -9601.187,E2 -9601.187} C_VEL
LIN {X 0,Y 435.34,Z 144.831,A -85,B 0,C 180,E1 -9603.8,E2 -9603.8} C_VEL
LIN {X 0,Y 441.535,Z 160.002,A -85,B 0,C 180,E1 -9604.467,E2 -9604.467} C_VEL
LIN {X 0,Y 443.735,Z 170.375,A -85,B 0,C 180,E1 -9604.786,E2 -9604.786} C_VEL
LIN {X 0,Y 442.039,Z 277.016,A -85,B 0,C 180,E1 -9606.548,E2 -9606.548} C_VEL
LIN {X 0,Y 441.488,Z 310.753,A -85,B 0,C 180,E1 -9607.137,E2 -9607.137} C_VEL
LIN {X 0,Y 440.936,Z 326.241,A -85,B 0,C 180,E1 -9607.594,E2 -9607.594} C_VEL
LIN {X 0,Y 440.307,Z 340.647,A -85,B 0,C 180,E1 -9608.203,E2 -9608.203} C_VEL
LIN {X 0,Y 439.976,Z 345.074,A -85,B 0,C 180,E1 -9608.428,E2 -9608.428} C_VEL
LIN {X 0,Y 438.869,Z 350.547,A -85,B 0,C 180,E1 -9608.687,E2 -9608.687} C_VEL
LIN {X 0,Y 435.543,Z 359.359,A -85,B 0,C 180,E1 -9609.101,E2 -9609.101} C_VEL
LIN {X 0,Y 432.272,Z 367.958,A -85,B 0,C 180,E1 -9609.589,E2 -9609.589} C_VEL
LIN {X 0,Y 431.243,Z 372.971,A -85,B 0,C 180,E1 -9609.968,E2 -9609.968} C_VEL
LIN {X 0,Y 430.054,Z 385.902,A -85,B 0,C 180,E1 -9611.172,E2 -9611.172} C_VEL
LIN {X 0,Y 428.999,Z 396.541,A -85,B 0,C 180,E1 -9612.358,E2 -9612.358} C_VEL
LIN {X 0,Y 427.949,Z 407.353,A -85,B 0,C 180,E1 -9613.789,E2 -9613.789} C_VEL
LIN {X 0,Y 426.858,Z 417.867,A -85,B 0,C 180,E1 -9615.458,E2 -9615.458} C_VEL
LIN {X 0,Y 426.033,Z 426.603,A -85,B 0,C 180,E1 -9617.132,E2 -9617.132} C_VEL
LIN {X 0,Y 425.503,Z 432.907,A -85,B 0,C 180,E1 -9618.568,E2 -9618.568} C_VEL
LIN {X 0,Y 424.926,Z 439.848,A -85,B 0,C 180,E1 -9620.48,E2 -9620.48} C_VEL
LIN {X 0,Y 424.553,Z 445.301,A -85,B 0,C 180,E1 -9622.39,E2 -9622.39} C_VEL
LIN {X 0,Y 424.353,Z 449.417,A -85,B 0,C 180,E1 -9624.297,E2 -9624.297} C_VEL
LIN {X 0,Y 424.155,Z 452.313,A -85,B 0,C 180,E1 -9626.2,E2 -9626.2} C_VEL
LIN {X 0,Y 424.149,Z 454.054,A -85,B 0,C 180,E1 -9628.101,E2 -9628.101} C_VEL
LIN {X 0,Y 424.084,Z 454.664,A -85,B 0,C 180,E1 -9630,E2 -9630} C_VEL
LIN {X 0,Y 424.149,Z 454.103,A -85,B 0,C 180,E1 -9631.899,E2 -9631.899} C_VEL
LIN {X 0,Y 424.154,Z 452.428,A -85,B 0,C 180,E1 -9633.8,E2 -9633.8} C_VEL
LIN {X 0,Y 424.348,Z 449.595,A -85,B 0,C 180,E1 -9635.703,E2 -9635.703} C_VEL
LIN {X 0,Y 424.541,Z 445.541,A -85,B 0,C 180,E1 -9637.61,E2 -9637.61} C_VEL
LIN {X 0,Y 424.916,Z 440.163,A -85,B 0,C 180,E1 -9639.52,E2 -9639.52} C_VEL
LIN {X 0,Y 425.489,Z 433.307,A -85,B 0,C 180,E1 -9641.432,E2 -9641.432} C_VEL
LIN {X 0,Y 426.109,Z 425.748,A -85,B 0,C 180,E1 -9643.149,E2 -9643.149} C_VEL
LIN {X 0,Y 426.943,Z 417.05,A -85,B 0,C 180,E1 -9644.783,E2 -9644.783} C_VEL
LIN {X 0,Y 427.88,Z 407.986,A -85,B 0,C 180,E1 -9646.214,E2 -9646.214} C_VEL
LIN {X 0,Y 428.979,Z 397.292,A -85,B 0,C 180,E1 -9647.643,E2 -9647.643} C_VEL
LIN {X 0,Y 430.076,Z 385.657,A -85,B 0,C 180,E1 -9648.948,E2 -9648.948} C_VEL
LIN {X 0,Y 431.288,Z 372.861,A -85,B 0,C 180,E1 -9650.136,E2 -9650.136} C_VEL
LIN {X 0,Y 432.308,Z 360.543,A -85,B 0,C 180,E1 -9651.081,E2 -9651.081} C_VEL
LIN {X 0,Y 433.407,Z 345.959,A -85,B 0,C 180,E1 -9651.974,E2 -9651.974} C_VEL
LIN {X 0,Y 434.181,Z 331.346,A -85,B 0,C 180,E1 -9652.668,E2 -9652.668} C_VEL
LIN {X 0,Y 434.816,Z 316.736,A -85,B 0,C 180,E1 -9653.171,E2 -9653.171} C_VEL
LIN {X 0,Y 435.243,Z 300.592,A -85,B 0,C 180,E1 -9653.525,E2 -9653.525} C_VEL
LIN {X 0,Y 437.295,Z 170.62,A -85,B 0,C 180,E1 -9655.709,E2 -9655.709} C_VEL
LIN {X 0,Y 434.861,Z 160.781,A -85,B 0,C 180,E1 -9656.042,E2 -9656.042} C_VEL
LIN {X 0,Y 428.106,Z 144.849,A -85,B 0,C 180,E1 -9656.808,E2 -9656.808} C_VEL
LIN {X 0,Y 425.268,Z 133.141,A -85,B 0,C 180,E1 -9659.366,E2 -9659.366} C_VEL
LIN {X 0,Y 425.266,Z 133.139,A -85,B 0,C 180,E1 -9662.559,E2 -9662.559} C_VEL
LIN {X 0,Y 425.29,Z 133.14,A -85,B 0,C 180,E1 -9665.337,E2 -9665.337} C_VEL
LIN {X 0,Y 425.265,Z 133.138,A -85,B 0,C 180,E1 -9668.903,E2 -9668.903} C_VEL
LIN {X 0,Y 425.263,Z 133.136,A -85,B 0,C 180,E1 -9671.954,E2 -9671.954} C_VEL
LIN {X 0,Y 425.284,Z 133.136,A -85,B 0,C 180,E1 -9675.284,E2 -9675.284} C_VEL
LIN {X 0,Y 425.248,Z 133.132,A -85,B 0,C 180,E1 -9678.618,E2 -9678.618} C_VEL
LIN {X 0,Y 425.277,Z 133.131,A -85,B 0,C 180,E1 -9681.099,E2 -9681.099} C_VEL
LIN {X 0,Y 425.294,Z 133.132,A -85,B 0,C 180,E1 -9684.663,E2 -9684.663} C_VEL
LIN {X 0,Y 425.254,Z 133.126,A -85,B 0,C 180,E1 -9688.072,E2 -9688.072} C_VEL
LIN {X 0,Y 425.293,Z 133.13,A -85,B 0,C 180,E1 -9691.365,E2 -9691.365} C_VEL
LIN {X 0,Y 425.262,Z 133.137,A -85,B 0,C 180,E1 -9694.552,E2 -9694.552} C_VEL
LIN {X 0,Y 425.293,Z 133.129,A -85,B 0,C 180,E1 -9697.73,E2 -9697.73} C_VEL
LIN {X 0,Y 425.362,Z 133.121,A -85,B 0,C 180,E1 -9700.704,E2 -9700.704} C_VEL
LIN {X 0,Y 425.325,Z 133.128,A -85,B 0,C 180,E1 -9703.686,E2 -9703.686} C_VEL
LIN {X 0,Y 425.397,Z 133.115,A -85,B 0,C 180,E1 -9707.096,E2 -9707.096} C_VEL
LIN {X 0,Y 425.397,Z 133.113,A -85,B 0,C 180,E1 -9710.49,E2 -9710.49} C_VEL
LIN {X 0,Y 425.479,Z 133.11,A -85,B 0,C 180,E1 -9713.36,E2 -9713.36} C_VEL
LIN {X 0,Y 425.349,Z 133.122,A -85,B 0,C 180,E1 -9715.261,E2 -9715.261} C_VEL
LIN {X 0,Y 425.568,Z 133.098,A -85,B 0,C 180,E1 -9718.107,E2 -9718.107} C_VEL
LIN {X 0,Y 425.614,Z 133.088,A -85,B 0,C 180,E1 -9720,E2 -9720} C_VEL
LIN {X 0,Y 425.538,Z 133.101,A -85,B 0,C 180,E1 -9722.84,E2 -9722.84} C_VEL
LIN {X 0,Y 425.534,Z 133.103,A -85,B 0,C 180,E1 -9725.687,E2 -9725.687} C_VEL
LIN {X 0,Y 425.411,Z 133.114,A -85,B 0,C 180,E1 -9728.551,E2 -9728.551} C_VEL
LIN {X 0,Y 425.415,Z 133.116,A -85,B 0,C 180,E1 -9732.402,E2 -9732.402} C_VEL
LIN {X 0,Y 425.39,Z 133.121,A -85,B 0,C 180,E1 -9736.312,E2 -9736.312} C_VEL
LIN {X 0,Y 425.331,Z 133.129,A -85,B 0,C 180,E1 -9739.635,E2 -9739.635} C_VEL
LIN {X 0,Y 425.306,Z 133.133,A -85,B 0,C 180,E1 -9743.365,E2 -9743.365} C_VEL
LIN {X 0,Y 425.303,Z 133.129,A -85,B 0,C 180,E1 -9746.498,E2 -9746.498} C_VEL
LIN {X 0,Y 425.288,Z 133.132,A -85,B 0,C 180,E1 -9749.72,E2 -9749.72} C_VEL
LIN {X 0,Y 425.283,Z 133.13,A -85,B 0,C 180,E1 -9753.048,E2 -9753.048} C_VEL
LIN {X 0,Y 425.283,Z 133.133,A -85,B 0,C 180,E1 -9755.928,E2 -9755.928} C_VEL
LIN {X 0,Y 425.283,Z 133.132,A -85,B 0,C 180,E1 -9759.04,E2 -9759.04} C_VEL
LIN {X 0,Y 425.291,Z 133.134,A -85,B 0,C 180,E1 -9761.958,E2 -9761.958} C_VEL
LIN {X 0,Y 425.286,Z 133.132,A -85,B 0,C 180,E1 -9765.283,E2 -9765.283} C_VEL
LIN {X 0,Y 425.276,Z 133.131,A -85,B 0,C 180,E1 -9768.621,E2 -9768.621} C_VEL
LIN {X 0,Y 425.311,Z 133.129,A -85,B 0,C 180,E1 -9771.102,E2 -9771.102} C_VEL
LIN {X 0,Y 425.3,Z 133.132,A -85,B 0,C 180,E1 -9774.664,E2 -9774.664} C_VEL
LIN {X 0,Y 425.292,Z 133.265,A -85,B 0,C 180,E1 -9777.405,E2 -9777.405} C_VEL
LIN {X 0,Y 429.034,Z 147.835,A -85,B 0,C 180,E1 -9780.249,E2 -9780.249} C_VEL
LIN {X 0,Y 431.305,Z 158.034,A -85,B 0,C 180,E1 -9782.145,E2 -9782.145} C_VEL
LIN {X 0,Y 430.761,Z 166.04,A -85,B 0,C 180,E1 -9783.436,E2 -9783.436} C_VEL
LIN {X 0,Y 436.921,Z 197.17,A -85,B 0,C 180,E1 -9784.393,E2 -9784.393} C_VEL
LIN {X 0,Y 435.384,Z 298.894,A -85,B 0,C 180,E1 -9786.105,E2 -9786.105} C_VEL
LIN {X 0,Y 434.753,Z 332.921,A -85,B 0,C 180,E1 -9786.7,E2 -9786.7} C_VEL
LIN {X 0,Y 434.058,Z 348.612,A -85,B 0,C 180,E1 -9787.157,E2 -9787.157} C_VEL
LIN {X 0,Y 433.22,Z 362.722,A -85,B 0,C 180,E1 -9787.745,E2 -9787.745} C_VEL
LIN {X 0,Y 432.188,Z 377.125,A -85,B 0,C 180,E1 -9788.538,E2 -9788.538} C_VEL
LIN {X 0,Y 431.014,Z 390.626,A -85,B 0,C 180,E1 -9789.477,E2 -9789.477} C_VEL
LIN {X 0,Y 429.781,Z 404.377,A -85,B 0,C 180,E1 -9790.662,E2 -9790.662} C_VEL
LIN {X 0,Y 428.528,Z 417.357,A -85,B 0,C 180,E1 -9792.03,E2 -9792.03} C_VEL
LIN {X 0,Y 427.388,Z 429.038,A -85,B 0,C 180,E1 -9793.521,E2 -9793.521} C_VEL
LIN {X 0,Y 426.468,Z 438.456,A -85,B 0,C 180,E1 -9794.956,E2 -9794.956} C_VEL
LIN {X 0,Y 425.603,Z 447.727,A -85,B 0,C 180,E1 -9796.633,E2 -9796.633} C_VEL
LIN {X 0,Y 425.064,Z 456.462,A -85,B 0,C 180,E1 -9798.556,E2 -9798.556} C_VEL
LIN {X 0,Y 424.514,Z 463.468,A -85,B 0,C 180,E1 -9800.47,E2 -9800.47} C_VEL
LIN {X 0,Y 424.306,Z 468.982,A -85,B 0,C 180,E1 -9802.385,E2 -9802.385} C_VEL
LIN {X 0,Y 424.139,Z 473.15,A -85,B 0,C 180,E1 -9804.294,E2 -9804.294} C_VEL
LIN {X 0,Y 424.051,Z 476.072,A -85,B 0,C 180,E1 -9806.199,E2 -9806.199} C_VEL
LIN {X 0,Y 424.124,Z 477.818,A -85,B 0,C 180,E1 -9808.101,E2 -9808.101} C_VEL
LIN {X 0,Y 424.082,Z 478.414,A -85,B 0,C 180,E1 -9810,E2 -9810} C_VEL
LIN {X 0,Y 424.124,Z 477.814,A -85,B 0,C 180,E1 -9811.899,E2 -9811.899} C_VEL
LIN {X 0,Y 424.051,Z 476.062,A -85,B 0,C 180,E1 -9813.801,E2 -9813.801} C_VEL
LIN {X 0,Y 424.151,Z 473.141,A -85,B 0,C 180,E1 -9815.706,E2 -9815.706} C_VEL
LIN {X 0,Y 424.306,Z 468.975,A -85,B 0,C 180,E1 -9817.615,E2 -9817.615} C_VEL
LIN {X 0,Y 424.514,Z 463.454,A -85,B 0,C 180,E1 -9819.529,E2 -9819.529} C_VEL
LIN {X 0,Y 425.046,Z 456.436,A -85,B 0,C 180,E1 -9821.444,E2 -9821.444} C_VEL
LIN {X 0,Y 425.603,Z 447.699,A -85,B 0,C 180,E1 -9823.367,E2 -9823.367} C_VEL
LIN {X 0,Y 426.468,Z 438.426,A -85,B 0,C 180,E1 -9825.044,E2 -9825.044} C_VEL
LIN {X 0,Y 427.348,Z 429,A -85,B 0,C 180,E1 -9826.48,E2 -9826.48} C_VEL
LIN {X 0,Y 428.494,Z 417.441,A -85,B 0,C 180,E1 -9827.956,E2 -9827.956} C_VEL
LIN {X 0,Y 429.611,Z 405.548,A -85,B 0,C 180,E1 -9829.222,E2 -9829.222} C_VEL
LIN {X 0,Y 430.876,Z 392.072,A -85,B 0,C 180,E1 -9830.405,E2 -9830.405} C_VEL
LIN {X 0,Y 432.054,Z 378.843,A -85,B 0,C 180,E1 -9831.344,E2 -9831.344} C_VEL
LIN {X 0,Y 433.033,Z 365.512,A -85,B 0,C 180,E1 -9832.106,E2 -9832.106} C_VEL
LIN {X 0,Y 433.898,Z 351.005,A -85,B 0,C 180,E1 -9832.747,E2 -9832.747} C_VEL
LIN {X 0,Y 434.575,Z 336.115,A -85,B 0,C 180,E1 -9833.216,E2 -9833.216} C_VEL
LIN {X 0,Y 435.082,Z 316.421,A -85,B 0,C 180,E1 -9833.597,E2 -9833.597} C_VEL
LIN {X 0,Y 437.003,Z 198.364,A -85,B 0,C 180,E1 -9835.574,E2 -9835.574} C_VEL
LIN {X 0,Y 432.259,Z 173.131,A -85,B 0,C 180,E1 -9836.329,E2 -9836.329} C_VEL
LIN {X 0,Y 430.691,Z 165.813,A -85,B 0,C 180,E1 -9836.573,E2 -9836.573} C_VEL
LIN {X 0,Y 431.3,Z 157.992,A -85,B 0,C 180,E1 -9837.854,E2 -9837.854} C_VEL
LIN {X 0,Y 428.633,Z 146.127,A -85,B 0,C 180,E1 -9840.064,E2 -9840.064} C_VEL
LIN {X 0,Y 425.291,Z 133.124,A -85,B 0,C 180,E1 -9842.619,E2 -9842.619} C_VEL
LIN {X 0,Y 425.3,Z 133.131,A -85,B 0,C 180,E1 -9845.336,E2 -9845.336} C_VEL
LIN {X 0,Y 425.301,Z 133.131,A -85,B 0,C 180,E1 -9849.044,E2 -9849.044} C_VEL
LIN {X 0,Y 425.275,Z 133.132,A -85,B 0,C 180,E1 -9852.653,E2 -9852.653} C_VEL
LIN {X 0,Y 425.262,Z 133.136,A -85,B 0,C 180,E1 -9856.044,E2 -9856.044} C_VEL
LIN {X 0,Y 425.275,Z 133.132,A -85,B 0,C 180,E1 -9858.622,E2 -9858.622} C_VEL
LIN {X 0,Y 425.298,Z 133.132,A -85,B 0,C 180,E1 -9861.101,E2 -9861.101} C_VEL
LIN {X 0,Y 425.299,Z 133.126,A -85,B 0,C 180,E1 -9864.664,E2 -9864.664} C_VEL
LIN {X 0,Y 425.265,Z 133.133,A -85,B 0,C 180,E1 -9868.073,E2 -9868.073} C_VEL
LIN {X 0,Y 425.332,Z 133.13,A -85,B 0,C 180,E1 -9871.368,E2 -9871.368} C_VEL
LIN {X 0,Y 425.284,Z 133.133,A -85,B 0,C 180,E1 -9874.554,E2 -9874.554} C_VEL
LIN {X 0,Y 425.285,Z 133.131,A -85,B 0,C 180,E1 -9876.634,E2 -9876.634} C_VEL
LIN {X 0,Y 425.297,Z 133.126,A -85,B 0,C 180,E1 -9879.695,E2 -9879.695} C_VEL
LIN {X 0,Y 425.335,Z 133.13,A -85,B 0,C 180,E1 -9882.697,E2 -9882.697} C_VEL
LIN {X 0,Y 425.348,Z 133.124,A -85,B 0,C 180,E1 -9885.65,E2 -9885.65} C_VEL
LIN {X 0,Y 425.352,Z 133.124,A -85,B 0,C 180,E1 -9888.564,E2 -9888.564} C_VEL
LIN {X 0,Y 425.41,Z 133.111,A -85,B 0,C 180,E1 -9891.449,E2 -9891.449} C_VEL
LIN {X 0,Y 425.534,Z 133.105,A -85,B 0,C 180,E1 -9894.313,E2 -9894.313} C_VEL
LIN {X 0,Y 425.574,Z 133.099,A -85,B 0,C 180,E1 -9898.107,E2 -9898.107} C_VEL
LIN {X 0,Y 425.511,Z 133.103,A -85,B 0,C 180,E1 -9900.946,E2 -9900.946} C_VEL
LIN {X 0,Y 425.518,Z 133.104,A -85,B 0,C 180,E1 -9902.84,E2 -9902.84} C_VEL
LIN {X 0,Y 425.482,Z 133.108,A -85,B 0,C 180,E1 -9906.474,E2 -9906.474} C_VEL
LIN {X 0,Y 425.397,Z 133.114,A -85,B 0,C 180,E1 -9909.51,E2 -9909.51} C_VEL
LIN {X 0,Y 425.396,Z 133.113,A -85,B 0,C 180,E1 -9912.904,E2 -9912.904} C_VEL
LIN {X 0,Y 425.319,Z 133.124,A -85,B 0,C 180,E1 -9916.585,E2 -9916.585} C_VEL
LIN {X 0,Y 425.33,Z 133.131,A -85,B 0,C 180,E1 -9919.635,E2 -9919.635} C_VEL
LIN {X 0,Y 425.289,Z 133.133,A -85,B 0,C 180,E1 -9922.339,E2 -9922.339} C_VEL
LIN {X 0,Y 425.261,Z 133.126,A -85,B 0,C 180,E1 -9925.448,E2 -9925.448} C_VEL
LIN {X 0,Y 425.308,Z 133.127,A -85,B 0,C 180,E1 -9928.86,E2 -9928.86} C_VEL
LIN {X 0,Y 425.264,Z 133.137,A -85,B 0,C 180,E1 -9931.927,E2 -9931.927} C_VEL
LIN {X 0,Y 425.295,Z 133.133,A -85,B 0,C 180,E1 -9935.336,E2 -9935.336} C_VEL
LIN {X 0,Y 425.279,Z 133.134,A -85,B 0,C 180,E1 -9938.901,E2 -9938.901} C_VEL
LIN {X 0,Y 425.257,Z 133.133,A -85,B 0,C 180,E1 -9942.655,E2 -9942.655} C_VEL
LIN {X 0,Y 425.286,Z 133.136,A -85,B 0,C 180,E1 -9945.283,E2 -9945.283} C_VEL
LIN {X 0,Y 425.248,Z 133.14,A -85,B 0,C 180,E1 -9948.618,E2 -9948.618} C_VEL
LIN {X 0,Y 425.276,Z 133.131,A -85,B 0,C 180,E1 -9951.099,E2 -9951.099} C_VEL
LIN {X 0,Y 425.291,Z 133.13,A -85,B 0,C 180,E1 -9954.663,E2 -9954.663} C_VEL
LIN {X 0,Y 425.247,Z 133.141,A -85,B 0,C 180,E1 -9958.071,E2 -9958.071} C_VEL
LIN {X 0,Y 425.281,Z 133.192,A -85,B 0,C 180,E1 -9960.795,E2 -9960.795} C_VEL
LIN {X 0,Y 428.163,Z 145.083,A -85,B 0,C 180,E1 -9963.326,E2 -9963.326} C_VEL
LIN {X 0,Y 435.363,Z 162.404,A -85,B 0,C 180,E1 -9964.118,E2 -9964.118} C_VEL
LIN {X 0,Y 437.302,Z 170.792,A -85,B 0,C 180,E1 -9964.392,E2 -9964.392} C_VEL
LIN {X 0,Y 435.622,Z 275.452,A -85,B 0,C 180,E1 -9966.15,E2 -9966.15} C_VEL
LIN {X 0,Y 434.968,Z 310.968,A -85,B 0,C 180,E1 -9966.775,E2 -9966.775} C_VEL
LIN {X 0,Y 434.377,Z 326.659,A -85,B 0,C 180,E1 -9967.245,E2 -9967.245} C_VEL
LIN {X 0,Y 433.707,Z 341.115,A -85,B 0,C 180,E1 -9967.869,E2 -9967.869} C_VEL
LIN {X 0,Y 432.674,Z 355.655,A -85,B 0,C 180,E1 -9968.688,E2 -9968.688} C_VEL
LIN {X 0,Y 431.626,Z 368.911,A -85,B 0,C 180,E1 -9969.632,E2 -9969.632} C_VEL
LIN {X 0,Y 431.243,Z 372.971,A -85,B 0,C 180,E1 -9969.968,E2 -9969.968} C_VEL
LIN {X 0,Y 430.171,Z 377.952,A -85,B 0,C 180,E1 -9970.369,E2 -9970.369} C_VEL
LIN {X 0,Y 426.69,Z 385.911,A -85,B 0,C 180,E1 -9971.006,E2 -9971.006} C_VEL
LIN {X 0,Y 423.187,Z 393.579,A -85,B 0,C 180,E1 -9971.713,E2 -9971.713} C_VEL
LIN {X 0,Y 422.09,Z 397.98,A -85,B 0,C 180,E1 -9972.219,E2 -9972.219} C_VEL
LIN {X 0,Y 420.919,Z 409.174,A -85,B 0,C 180,E1 -9973.759,E2 -9973.759} C_VEL
LIN {X 0,Y 419.794,Z 419.414,A -85,B 0,C 180,E1 -9975.456,E2 -9975.456} C_VEL
LIN {X 0,Y 419.028,Z 427.517,A -85,B 0,C 180,E1 -9977.072,E2 -9977.072} C_VEL
LIN {X 0,Y 418.31,Z 434.982,A -85,B 0,C 180,E1 -9978.86,E2 -9978.86} C_VEL
LIN {X 0,Y 417.793,Z 441.539,A -85,B 0,C 180,E1 -9980.804,E2 -9980.804} C_VEL
LIN {X 0,Y 417.431,Z 446.665,A -85,B 0,C 180,E1 -9982.746,E2 -9982.746} C_VEL
LIN {X 0,Y 417.285,Z 449.617,A -85,B 0,C 180,E1 -9984.2,E2 -9984.2} C_VEL
LIN {X 0,Y 417.067,Z 452.512,A -85,B 0,C 180,E1 -9986.135,E2 -9986.135} C_VEL
LIN {X 0,Y 417.077,Z 454.252,A -85,B 0,C 180,E1 -9988.069,E2 -9988.069} C_VEL
LIN {X 0,Y 417.003,Z 454.862,A -85,B 0,C 180,E1 -9990,E2 -9990} C_VEL
LIN {X 0,Y 417.078,Z 454.301,A -85,B 0,C 180,E1 -9991.931,E2 -9991.931} C_VEL
LIN {X 0,Y 417.066,Z 452.627,A -85,B 0,C 180,E1 -9993.865,E2 -9993.865} C_VEL
LIN {X 0,Y 417.28,Z 449.793,A -85,B 0,C 180,E1 -9995.8,E2 -9995.8} C_VEL
LIN {X 0,Y 417.48,Z 445.739,A -85,B 0,C 180,E1 -9997.74,E2 -9997.74} C_VEL
LIN {X 0,Y 417.882,Z 440.361,A -85,B 0,C 180,E1 -9999.682,E2 -9999.682} C_VEL
LIN {X 0,Y 418.523,Z 433.505,A -85,B 0,C 180,E1 -10001.625,E2 -10001.625} C_VEL
LIN {X 0,Y 419.201,Z 425.338,A -85,B 0,C 180,E1 -10003.496,E2 -10003.496} C_VEL
LIN {X 0,Y 420.205,Z 415.845,A -85,B 0,C 180,E1 -10005.273,E2 -10005.273} C_VEL
LIN {X 0,Y 421.239,Z 406.565,A -85,B 0,C 180,E1 -10006.726,E2 -10006.726} C_VEL
LIN {X 0,Y 422.411,Z 395.546,A -85,B 0,C 180,E1 -10008.177,E2 -10008.177} C_VEL
LIN {X 0,Y 423.537,Z 383.477,A -85,B 0,C 180,E1 -10009.509,E2 -10009.509} C_VEL
LIN {X 0,Y 424.877,Z 370.216,A -85,B 0,C 180,E1 -10010.706,E2 -10010.706} C_VEL
LIN {X 0,Y 426.007,Z 357.213,A -85,B 0,C 180,E1 -10011.662,E2 -10011.662} C_VEL
LIN {X 0,Y 427.021,Z 343.663,A -85,B 0,C 180,E1 -10012.461,E2 -10012.461} C_VEL
LIN {X 0,Y 427.761,Z 329.24,A -85,B 0,C 180,E1 -10013.124,E2 -10013.124} C_VEL
LIN {X 0,Y 428.412,Z 313.504,A -85,B 0,C 180,E1 -10013.634,E2 -10013.634} C_VEL
LIN {X 0,Y 428.896,Z 293.615,A -85,B 0,C 180,E1 -10014.023,E2 -10014.023} C_VEL
LIN {X 0,Y 430.941,Z 172.11,A -85,B 0,C 180,E1 -10016.092,E2 -10016.092} C_VEL
LIN {X 0,Y 428.902,Z 163.713,A -85,B 0,C 180,E1 -10016.381,E2 -10016.381} C_VEL
LIN {X 0,Y 420.969,Z 145.178,A -85,B 0,C 180,E1 -10017.277,E2 -10017.277} C_VEL
LIN {X 0,Y 418.231,Z 134.016,A -85,B 0,C 180,E1 -10019.752,E2 -10019.752} C_VEL
LIN {X 0,Y 418.241,Z 134.016,A -85,B 0,C 180,E1 -10022.84,E2 -10022.84} C_VEL
LIN {X 0,Y 418.238,Z 134.012,A -85,B 0,C 180,E1 -10026.236,E2 -10026.236} C_VEL
LIN {X 0,Y 418.194,Z 134.012,A -85,B 0,C 180,E1 -10029.689,E2 -10029.689} C_VEL
LIN {X 0,Y 418.206,Z 134.016,A -85,B 0,C 180,E1 -10032.317,E2 -10032.317} C_VEL
LIN {X 0,Y 418.235,Z 134.016,A -85,B 0,C 180,E1 -10035.108,E2 -10035.108} C_VEL
LIN {X 0,Y 418.219,Z 134.003,A -85,B 0,C 180,E1 -10037.764,E2 -10037.764} C_VEL
LIN {X 0,Y 418.235,Z 134.004,A -85,B 0,C 180,E1 -10041.556,E2 -10041.556} C_VEL
LIN {X 0,Y 418.251,Z 134.011,A -85,B 0,C 180,E1 -10045.158,E2 -10045.158} C_VEL
LIN {X 0,Y 418.241,Z 134.002,A -85,B 0,C 180,E1 -10047.471,E2 -10047.471} C_VEL
LIN {X 0,Y 418.259,Z 134.009,A -85,B 0,C 180,E1 -10050.899,E2 -10050.899} C_VEL
LIN {X 0,Y 418.22,Z 134.011,A -85,B 0,C 180,E1 -10054.092,E2 -10054.092} C_VEL
LIN {X 0,Y 418.23,Z 134.008,A -85,B 0,C 180,E1 -10057.263,E2 -10057.263} C_VEL
LIN {X 0,Y 418.285,Z 134.007,A -85,B 0,C 180,E1 -10060.364,E2 -10060.364} C_VEL
LIN {X 0,Y 418.281,Z 134.004,A -85,B 0,C 180,E1 -10063.403,E2 -10063.403} C_VEL
LIN {X 0,Y 418.349,Z 133.993,A -85,B 0,C 180,E1 -10066.999,E2 -10066.999} C_VEL
LIN {X 0,Y 418.338,Z 133.993,A -85,B 0,C 180,E1 -10070.328,E2 -10070.328} C_VEL
LIN {X 0,Y 418.444,Z 133.985,A -85,B 0,C 180,E1 -10073.248,E2 -10073.248} C_VEL
LIN {X 0,Y 418.319,Z 133.997,A -85,B 0,C 180,E1 -10075.181,E2 -10075.181} C_VEL
LIN {X 0,Y 418.536,Z 133.974,A -85,B 0,C 180,E1 -10078.075,E2 -10078.075} C_VEL
LIN {X 0,Y 418.565,Z 133.966,A -85,B 0,C 180,E1 -10080,E2 -10080} C_VEL
LIN {X 0,Y 418.493,Z 133.979,A -85,B 0,C 180,E1 -10082.888,E2 -10082.888} C_VEL
LIN {X 0,Y 418.492,Z 133.982,A -85,B 0,C 180,E1 -10085.783,E2 -10085.783} C_VEL
LIN {X 0,Y 418.38,Z 133.991,A -85,B 0,C 180,E1 -10088.695,E2 -10088.695} C_VEL
LIN {X 0,Y 418.317,Z 134.004,A -85,B 0,C 180,E1 -10091.631,E2 -10091.631} C_VEL
LIN {X 0,Y 418.302,Z 133.999,A -85,B 0,C 180,E1 -10094.597,E2 -10094.597} C_VEL
LIN {X 0,Y 418.281,Z 134.001,A -85,B 0,C 180,E1 -10097.604,E2 -10097.604} C_VEL
LIN {X 0,Y 418.252,Z 134.013,A -85,B 0,C 180,E1 -10100.663,E2 -10100.663} C_VEL
LIN {X 0,Y 418.286,Z 134.005,A -85,B 0,C 180,E1 -10103.781,E2 -10103.781} C_VEL
LIN {X 0,Y 418.268,Z 134.008,A -85,B 0,C 180,E1 -10107.058,E2 -10107.058} C_VEL
LIN {X 0,Y 418.244,Z 134.011,A -85,B 0,C 180,E1 -10110.272,E2 -10110.272} C_VEL
LIN {X 0,Y 418.249,Z 134.003,A -85,B 0,C 180,E1 -10113.677,E2 -10113.677} C_VEL
LIN {X 0,Y 418.241,Z 134.009,A -85,B 0,C 180,E1 -10117.224,E2 -10117.224} C_VEL
LIN {X 0,Y 418.246,Z 134.007,A -85,B 0,C 180,E1 -10119.682,E2 -10119.682} C_VEL
LIN {X 0,Y 418.231,Z 134.013,A -85,B 0,C 180,E1 -10122.321,E2 -10122.321} C_VEL
LIN {X 0,Y 418.237,Z 134.011,A -85,B 0,C 180,E1 -10125.108,E2 -10125.108} C_VEL
LIN {X 0,Y 418.241,Z 134.011,A -85,B 0,C 180,E1 -10127.767,E2 -10127.767} C_VEL
LIN {X 0,Y 418.256,Z 134.005,A -85,B 0,C 180,E1 -10130.619,E2 -10130.619} C_VEL
LIN {X 0,Y 418.244,Z 134.012,A -85,B 0,C 180,E1 -10133.976,E2 -10133.976} C_VEL
LIN {X 0,Y 418.281,Z 134.154,A -85,B 0,C 180,E1 -10136.989,E2 -10136.989} C_VEL
LIN {X 0,Y 422.179,Z 149.47,A -85,B 0,C 180,E1 -10140.039,E2 -10140.039} C_VEL
LIN {X 0,Y 424.437,Z 159.392,A -85,B 0,C 180,E1 -10141.923,E2 -10141.923} C_VEL
LIN {X 0,Y 424.075,Z 165.664,A -85,B 0,C 180,E1 -10142.978,E2 -10142.978} C_VEL
LIN {X 0,Y 430.052,Z 195.708,A -85,B 0,C 180,E1 -10143.93,E2 -10143.93} C_VEL
LIN {X 0,Y 430.592,Z 199.96,A -85,B 0,C 180,E1 -10144.042,E2 -10144.042} C_VEL
LIN {X 0,Y 428.285,Z 331.431,A -85,B 0,C 180,E1 -10146.294,E2 -10146.294} C_VEL
LIN {X 0,Y 427.605,Z 346.965,A -85,B 0,C 180,E1 -10146.736,E2 -10146.736} C_VEL
LIN {X 0,Y 426.711,Z 360.827,A -85,B 0,C 180,E1 -10147.303,E2 -10147.303} C_VEL
LIN {X 0,Y 425.707,Z 374.94,A -85,B 0,C 180,E1 -10148.067,E2 -10148.067} C_VEL
LIN {X 0,Y 424.454,Z 388.844,A -85,B 0,C 180,E1 -10149.019,E2 -10149.019} C_VEL
LIN {X 0,Y 423.261,Z 401.588,A -85,B 0,C 180,E1 -10150.099,E2 -10150.099} C_VEL
LIN {X 0,Y 422.065,Z 413.405,A -85,B 0,C 180,E1 -10151.304,E2 -10151.304} C_VEL
LIN {X 0,Y 420.911,Z 425.278,A -85,B 0,C 180,E1 -10152.76,E2 -10152.76} C_VEL
LIN {X 0,Y 419.816,Z 435.269,A -85,B 0,C 180,E1 -10154.214,E2 -10154.214} C_VEL
LIN {X 0,Y 418.856,Z 445.048,A -85,B 0,C 180,E1 -10155.919,E2 -10155.919} C_VEL
LIN {X 0,Y 418.215,Z 453.214,A -85,B 0,C 180,E1 -10157.628,E2 -10157.628} C_VEL
LIN {X 0,Y 417.684,Z 459.964,A -85,B 0,C 180,E1 -10159.334,E2 -10159.334} C_VEL
LIN {X 0,Y 417.3,Z 466.201,A -85,B 0,C 180,E1 -10161.282,E2 -10161.282} C_VEL
LIN {X 0,Y 417.147,Z 471.028,A -85,B 0,C 180,E1 -10163.227,E2 -10163.227} C_VEL
LIN {X 0,Y 417.022,Z 474.564,A -85,B 0,C 180,E1 -10165.166,E2 -10165.166} C_VEL
LIN {X 0,Y 417.006,Z 476.891,A -85,B 0,C 180,E1 -10167.102,E2 -10167.102} C_VEL
LIN {X 0,Y 417.007,Z 478.062,A -85,B 0,C 180,E1 -10169.034,E2 -10169.034} C_VEL
LIN {X 0,Y 417.007,Z 478.06,A -85,B 0,C 180,E1 -10170.966,E2 -10170.966} C_VEL
LIN {X 0,Y 417.006,Z 476.883,A -85,B 0,C 180,E1 -10172.898,E2 -10172.898} C_VEL
LIN {X 0,Y 417.025,Z 474.553,A -85,B 0,C 180,E1 -10174.834,E2 -10174.834} C_VEL
LIN {X 0,Y 417.155,Z 471.019,A -85,B 0,C 180,E1 -10176.773,E2 -10176.773} C_VEL
LIN {X 0,Y 417.3,Z 466.19,A -85,B 0,C 180,E1 -10178.718,E2 -10178.718} C_VEL
LIN {X 0,Y 417.682,Z 459.941,A -85,B 0,C 180,E1 -10180.666,E2 -10180.666} C_VEL
LIN {X 0,Y 418.212,Z 453.186,A -85,B 0,C 180,E1 -10182.372,E2 -10182.372} C_VEL
LIN {X 0,Y 418.999,Z 443.755,A -85,B 0,C 180,E1 -10184.324,E2 -10184.324} C_VEL
LIN {X 0,Y 419.938,Z 433.71,A -85,B 0,C 180,E1 -10186.03,E2 -10186.03} C_VEL
LIN {X 0,Y 421.212,Z 422.324,A -85,B 0,C 180,E1 -10187.626,E2 -10187.626} C_VEL
LIN {X 0,Y 422.386,Z 410.057,A -85,B 0,C 180,E1 -10189.059,E2 -10189.059} C_VEL
LIN {X 0,Y 423.638,Z 397.595,A -85,B 0,C 180,E1 -10190.262,E2 -10190.262} C_VEL
LIN {X 0,Y 424.917,Z 383.949,A -85,B 0,C 180,E1 -10191.338,E2 -10191.338} C_VEL
LIN {X 0,Y 426.111,Z 369.817,A -85,B 0,C 180,E1 -10192.23,E2 -10192.23} C_VEL
LIN {X 0,Y 427.158,Z 354.426,A -85,B 0,C 180,E1 -10192.975,E2 -10192.975} C_VEL
LIN {X 0,Y 427.947,Z 339.333,A -85,B 0,C 180,E1 -10193.501,E2 -10193.501} C_VEL
